LIN {X 0,Y 325.912,Z 530.757,A -85,B 0,C 180,E1 14086.323,E2 14086.323} C_VEL
LIN {X 0,Y 331.424,Z 417.148,A -85,B 0,C 180,E1 14083.968,E2 14083.968} C_VEL
LIN {X 0,Y 322.089,Z 400.841,A -85,B 0,C 180,E1 14081.452,E2 14081.452} C_VEL
LIN {X 0,Y 313.138,Z 386.861,A -85,B 0,C 180,E1 14078.803,E2 14078.803} C_VEL
LIN {X 0,Y 303.548,Z 373.217,A -85,B 0,C 180,E1 14075.606,E2 14075.606} C_VEL
LIN {X 0,Y 293.892,Z 360.856,A -85,B 0,C 180,E1 14071.883,E2 14071.883} C_VEL
LIN {X 0,Y 289.242,Z 355.015,A -85,B 0,C 180,E1 14069.74,E2 14069.74} C_VEL
LIN {X 0,Y 286.141,Z 348.999,A -85,B 0,C 180,E1 14066.345,E2 14066.345} C_VEL
LIN {X 0,Y 283.721,Z 344.309,A -85,B 0,C 180,E1 14063.248,E2 14063.248} C_VEL
LIN {X 0,Y 281.408,Z 340.402,A -85,B 0,C 180,E1 14059.944,E2 14059.944} C_VEL
LIN {X 0,Y 280.7,Z 339.051,A -85,B 0,C 180,E1 14058.699,E2 14058.699} C_VEL
LIN {X 0,Y 277.789,Z 333.962,A -85,B 0,C 180,E1 14052.05,E2 14052.05} C_VEL
LIN {X 0,Y 276.387,Z 332.628,A -85,B 0,C 180,E1 14046.439,E2 14046.439} C_VEL
LIN {X 0,Y 276.572,Z 332.801,A -85,B 0,C 180,E1 14041.243,E2 14041.243} C_VEL
LIN {X 0,Y 278.076,Z 334.319,A -85,B 0,C 180,E1 14036.29,E2 14036.29} C_VEL
LIN {X 0,Y 281.635,Z 340.034,A -85,B 0,C 180,E1 14029.362,E2 14029.362} C_VEL
LIN {X 0,Y 283.845,Z 344.262,A -85,B 0,C 180,E1 14026.141,E2 14026.141} C_VEL
LIN {X 0,Y 284.804,Z 345.431,A -85,B 0,C 180,E1 14025.151,E2 14025.151} C_VEL
LIN {X 0,Y 287.071,Z 349.665,A -85,B 0,C 180,E1 14022.571,E2 14022.571} C_VEL
LIN {X 0,Y 287.875,Z 350.984,A -85,B 0,C 180,E1 14021.785,E2 14021.785} C_VEL
LIN {X 0,Y 290.746,Z 356.23,A -85,B 0,C 180,E1 14019.044,E2 14019.044} C_VEL
LIN {X 0,Y 293.325,Z 361.286,A -85,B 0,C 180,E1 14016.709,E2 14016.709} C_VEL
LIN {X 0,Y 297.429,Z 368.871,A -85,B 0,C 180,E1 14013.658,E2 14013.658} C_VEL
LIN {X 0,Y 299.486,Z 372.66,A -85,B 0,C 180,E1 14012.405,E2 14012.405} C_VEL
LIN {X 0,Y 308.932,Z 386.315,A -85,B 0,C 180,E1 14009.029,E2 14009.029} C_VEL
LIN {X 0,Y 317.812,Z 400.47,A -85,B 0,C 180,E1 14006.216,E2 14006.216} C_VEL
LIN {X 0,Y 327.251,Z 417.04,A -85,B 0,C 180,E1 14003.513,E2 14003.513} C_VEL
LIN {X 0,Y 331.466,Z 425.611,A -85,B 0,C 180,E1 14002.357,E2 14002.357} C_VEL
LIN {X 0,Y 331.933,Z 439.03,A -85,B 0,C 180,E1 14001.807,E2 14001.807} C_VEL
LIN {X 0,Y 321.091,Z 624.81,A -85,B 0,C 180,E1 13997.585,E2 13997.585} C_VEL
LIN {X 0,Y 318.521,Z 646.616,A -85,B 0,C 180,E1 13996.819,E2 13996.819} C_VEL
LIN {X 0,Y 314.877,Z 667.549,A -85,B 0,C 180,E1 13995.793,E2 13995.793} C_VEL
LIN {X 0,Y 310.481,Z 687.705,A -85,B 0,C 180,E1 13994.459,E2 13994.459} C_VEL
LIN {X 0,Y 305.511,Z 707.389,A -85,B 0,C 180,E1 13992.755,E2 13992.755} C_VEL
LIN {X 0,Y 300.341,Z 725.782,A -85,B 0,C 180,E1 13990.729,E2 13990.729} C_VEL
LIN {X 0,Y 295.179,Z 742.727,A -85,B 0,C 180,E1 13988.414,E2 13988.414} C_VEL
LIN {X 0,Y 290.123,Z 758.694,A -85,B 0,C 180,E1 13985.742,E2 13985.742} C_VEL
LIN {X 0,Y 285.541,Z 773.07,A -85,B 0,C 180,E1 13982.819,E2 13982.819} C_VEL
LIN {X 0,Y 281.238,Z 787.006,A -85,B 0,C 180,E1 13979.38,E2 13979.38} C_VEL
LIN {X 0,Y 277.714,Z 799.537,A -85,B 0,C 180,E1 13975.596,E2 13975.596} C_VEL
LIN {X 0,Y 275.265,Z 809.934,A -85,B 0,C 180,E1 13971.746,E2 13971.746} C_VEL
LIN {X 0,Y 273.777,Z 818.455,A -85,B 0,C 180,E1 13967.864,E2 13967.864} C_VEL
LIN {X 0,Y 273.13,Z 825.558,A -85,B 0,C 180,E1 13963.765,E2 13963.765} C_VEL
LIN {X 0,Y 273.196,Z 830.779,A -85,B 0,C 180,E1 13959.692,E2 13959.692} C_VEL
LIN {X 0,Y 273.612,Z 834.096,A -85,B 0,C 180,E1 13955.873,E2 13955.873} C_VEL
LIN {X 0,Y 273.979,Z 835.824,A -85,B 0,C 180,E1 13952.301,E2 13952.301} C_VEL
LIN {X 0,Y 274.057,Z 836.01,A -85,B 0,C 180,E1 13948.955,E2 13948.955} C_VEL
LIN {X 0,Y 273.763,Z 834.896,A -85,B 0,C 180,E1 13945.391,E2 13945.391} C_VEL
LIN {X 0,Y 273.337,Z 832.235,A -85,B 0,C 180,E1 13941.798,E2 13941.798} C_VEL
LIN {X 0,Y 273.084,Z 827.633,A -85,B 0,C 180,E1 13937.74,E2 13937.74} C_VEL
LIN {X 0,Y 273.452,Z 821.244,A -85,B 0,C 180,E1 13933.648,E2 13933.648} C_VEL
LIN {X 0,Y 274.661,Z 812.965,A -85,B 0,C 180,E1 13929.546,E2 13929.546} C_VEL
LIN {X 0,Y 276.918,Z 802.631,A -85,B 0,C 180,E1 13925.467,E2 13925.467} C_VEL
LIN {X 0,Y 280.149,Z 790.716,A -85,B 0,C 180,E1 13921.662,E2 13921.662} C_VEL
LIN {X 0,Y 284.213,Z 777.257,A -85,B 0,C 180,E1 13918.151,E2 13918.151} C_VEL
LIN {X 0,Y 288.798,Z 762.744,A -85,B 0,C 180,E1 13915.043,E2 13915.043} C_VEL
LIN {X 0,Y 293.673,Z 747.357,A -85,B 0,C 180,E1 13912.329,E2 13912.329} C_VEL
LIN {X 0,Y 298.826,Z 730.575,A -85,B 0,C 180,E1 13909.903,E2 13909.903} C_VEL
LIN {X 0,Y 304.127,Z 712.146,A -85,B 0,C 180,E1 13907.755,E2 13907.755} C_VEL
LIN {X 0,Y 309.042,Z 693.226,A -85,B 0,C 180,E1 13906.004,E2 13906.004} C_VEL
LIN {X 0,Y 313.618,Z 673.067,A -85,B 0,C 180,E1 13904.559,E2 13904.559} C_VEL
LIN {X 0,Y 317.514,Z 652.33,A -85,B 0,C 180,E1 13903.454,E2 13903.454} C_VEL
LIN {X 0,Y 320.333,Z 631.352,A -85,B 0,C 180,E1 13902.639,E2 13902.639} C_VEL
LIN {X 0,Y 322.11,Z 608.021,A -85,B 0,C 180,E1 13902.015,E2 13902.015} C_VEL
LIN {X 0,Y 331.889,Z 436.421,A -85,B 0,C 180,E1 13898.133,E2 13898.133} C_VEL
LIN {X 0,Y 331.118,Z 424.68,A -85,B 0,C 180,E1 13897.587,E2 13897.587} C_VEL
LIN {X 0,Y 322.829,Z 409.225,A -85,B 0,C 180,E1 13895.31,E2 13895.31} C_VEL
LIN {X 0,Y 314.205,Z 394.789,A -85,B 0,C 180,E1 13892.749,E2 13892.749} C_VEL
LIN {X 0,Y 306.355,Z 382.678,A -85,B 0,C 180,E1 13890.173,E2 13890.173} C_VEL
LIN {X 0,Y 298.711,Z 371.628,A -85,B 0,C 180,E1 13887.349,E2 13887.349} C_VEL
LIN {X 0,Y 294.503,Z 363.438,A -85,B 0,C 180,E1 13884.255,E2 13884.255} C_VEL
LIN {X 0,Y 291.847,Z 358.564,A -85,B 0,C 180,E1 13882.139,E2 13882.139} C_VEL
LIN {X 0,Y 289.754,Z 354.487,A -85,B 0,C 180,E1 13880.186,E2 13880.186} C_VEL
LIN {X 0,Y 287.159,Z 349.76,A -85,B 0,C 180,E1 13877.633,E2 13877.633} C_VEL
LIN {X 0,Y 284.83,Z 345.563,A -85,B 0,C 180,E1 13875.056,E2 13875.056} C_VEL
LIN {X 0,Y 281.786,Z 340.679,A -85,B 0,C 180,E1 13871.253,E2 13871.253} C_VEL
LIN {X 0,Y 281.192,Z 339.431,A -85,B 0,C 180,E1 13870.241,E2 13870.241} C_VEL
LIN {X 0,Y 277.823,Z 333.98,A -85,B 0,C 180,E1 13863.507,E2 13863.507} C_VEL
LIN {X 0,Y 276.215,Z 332.418,A -85,B 0,C 180,E1 13857.505,E2 13857.505} C_VEL
LIN {X 0,Y 276.38,Z 332.578,A -85,B 0,C 180,E1 13852.098,E2 13852.098} C_VEL
LIN {X 0,Y 277.952,Z 334.225,A -85,B 0,C 180,E1 13846.901,E2 13846.901} C_VEL
LIN {X 0,Y 281.193,Z 339.671,A -85,B 0,C 180,E1 13840.257,E2 13840.257} C_VEL
LIN {X 0,Y 283.306,Z 343.892,A -85,B 0,C 180,E1 13836.936,E2 13836.936} C_VEL
LIN {X 0,Y 284.176,Z 345.216,A -85,B 0,C 180,E1 13835.911,E2 13835.911} C_VEL
LIN {X 0,Y 286.766,Z 350.132,A -85,B 0,C 180,E1 13832.757,E2 13832.757} C_VEL
LIN {X 0,Y 289.262,Z 355.103,A -85,B 0,C 180,E1 13830.034,E2 13830.034} C_VEL
LIN {X 0,Y 295.268,Z 362.715,A -85,B 0,C 180,E1 13827.366,E2 13827.366} C_VEL
LIN {X 0,Y 303.925,Z 373.809,A -85,B 0,C 180,E1 13824.097,E2 13824.097} C_VEL
LIN {X 0,Y 313.853,Z 387.94,A -85,B 0,C 180,E1 13820.833,E2 13820.833} C_VEL
LIN {X 0,Y 323.057,Z 402.598,A -85,B 0,C 180,E1 13818.136,E2 13818.136} C_VEL
LIN {X 0,Y 331.436,Z 417.301,A -85,B 0,C 180,E1 13815.892,E2 13815.892} C_VEL
LIN {X 0,Y 324.029,Z 570.746,A -85,B 0,C 180,E1 13812.693,E2 13812.693} C_VEL
LIN {X 0,Y 322.622,Z 590.161,A -85,B 0,C 180,E1 13812.013,E2 13812.013} C_VEL
LIN {X 0,Y 320.358,Z 608.777,A -85,B 0,C 180,E1 13811.069,E2 13811.069} C_VEL
LIN {X 0,Y 317.4,Z 626.429,A -85,B 0,C 180,E1 13809.869,E2 13809.869} C_VEL
LIN {X 0,Y 313.615,Z 644.125,A -85,B 0,C 180,E1 13808.322,E2 13808.322} C_VEL
LIN {X 0,Y 309.308,Z 660.695,A -85,B 0,C 180,E1 13806.497,E2 13806.497} C_VEL
LIN {X 0,Y 304.53,Z 676.538,A -85,B 0,C 180,E1 13804.313,E2 13804.313} C_VEL
LIN {X 0,Y 299.564,Z 691.068,A -85,B 0,C 180,E1 13801.826,E2 13801.826} C_VEL
LIN {X 0,Y 294.635,Z 704.227,A -85,B 0,C 180,E1 13799.03,E2 13799.03} C_VEL
LIN {X 0,Y 289.962,Z 715.814,A -85,B 0,C 180,E1 13795.971,E2 13795.971} C_VEL
LIN {X 0,Y 285.729,Z 725.888,A -85,B 0,C 180,E1 13792.638,E2 13792.638} C_VEL
LIN {X 0,Y 282.058,Z 734.454,A -85,B 0,C 180,E1 13789.033,E2 13789.033} C_VEL
LIN {X 0,Y 279.071,Z 741.482,A -85,B 0,C 180,E1 13785.161,E2 13785.161} C_VEL
LIN {X 0,Y 276.972,Z 746.671,A -85,B 0,C 180,E1 13781.241,E2 13781.241} C_VEL
LIN {X 0,Y 275.562,Z 750.342,A -85,B 0,C 180,E1 13777.086,E2 13777.086} C_VEL
LIN {X 0,Y 274.872,Z 752.306,A -85,B 0,C 180,E1 13772.919,E2 13772.919} C_VEL
LIN {X 0,Y 274.762,Z 752.649,A -85,B 0,C 180,E1 13768.749,E2 13768.749} C_VEL
LIN {X 0,Y 275.198,Z 751.384,A -85,B 0,C 180,E1 13764.572,E2 13764.572} C_VEL
LIN {X 0,Y 276.288,Z 748.463,A -85,B 0,C 180,E1 13760.418,E2 13760.418} C_VEL
LIN {X 0,Y 278.158,Z 743.76,A -85,B 0,C 180,E1 13756.277,E2 13756.277} C_VEL
LIN {X 0,Y 280.792,Z 737.489,A -85,B 0,C 180,E1 13752.382,E2 13752.382} C_VEL
LIN {X 0,Y 284.139,Z 729.734,A -85,B 0,C 180,E1 13748.75,E2 13748.75} C_VEL
LIN {X 0,Y 288.037,Z 720.554,A -85,B 0,C 180,E1 13745.384,E2 13745.384} C_VEL
LIN {X 0,Y 292.411,Z 709.978,A -85,B 0,C 180,E1 13742.289,E2 13742.289} C_VEL
LIN {X 0,Y 297.09,Z 698.005,A -85,B 0,C 180,E1 13739.458,E2 13739.458} C_VEL
LIN {X 0,Y 302.111,Z 684.038,A -85,B 0,C 180,E1 13736.789,E2 13736.789} C_VEL
LIN {X 0,Y 307.017,Z 668.867,A -85,B 0,C 180,E1 13734.458,E2 13734.458} C_VEL
LIN {X 0,Y 311.62,Z 652.509,A -85,B 0,C 180,E1 13732.438,E2 13732.438} C_VEL
LIN {X 0,Y 315.588,Z 635.868,A -85,B 0,C 180,E1 13730.799,E2 13730.799} C_VEL
LIN {X 0,Y 318.977,Z 618.266,A -85,B 0,C 180,E1 13729.428,E2 13729.428} C_VEL
LIN {X 0,Y 321.711,Z 599.435,A -85,B 0,C 180,E1 13728.312,E2 13728.312} C_VEL
LIN {X 0,Y 323.578,Z 579.916,A -85,B 0,C 180,E1 13727.482,E2 13727.482} C_VEL
LIN {X 0,Y 324.743,Z 555.923,A -85,B 0,C 180,E1 13726.846,E2 13726.846} C_VEL
LIN {X 0,Y 325.912,Z 530.757,A -85,B 0,C 180,E1 13726.323,E2 13726.323} C_VEL
LIN {X 0,Y 325.598,Z 523.167,A -85,B 0,C 180,E1 13726.039,E2 13726.039} C_VEL
LIN {X 0,Y 322.366,Z 503.342,A -85,B 0,C 180,E1 13724.812,E2 13724.812} C_VEL
LIN {X 0,Y 322.193,Z 496.817,A -85,B 0,C 180,E1 13724.576,E2 13724.576} C_VEL
LIN {X 0,Y 326.056,Z 420.531,A -85,B 0,C 180,E1 13722.97,E2 13722.97} C_VEL
LIN {X 0,Y 317.729,Z 405.913,A -85,B 0,C 180,E1 13720.619,E2 13720.619} C_VEL
LIN {X 0,Y 309.549,Z 392.937,A -85,B 0,C 180,E1 13718.093,E2 13718.093} C_VEL
LIN {X 0,Y 300.513,Z 379.839,A -85,B 0,C 180,E1 13714.968,E2 13714.968} C_VEL
LIN {X 0,Y 291.185,Z 367.626,A -85,B 0,C 180,E1 13711.232,E2 13711.232} C_VEL
LIN {X 0,Y 285.424,Z 360.648,A -85,B 0,C 180,E1 13708.566,E2 13708.566} C_VEL
LIN {X 0,Y 281.908,Z 356.155,A -85,B 0,C 180,E1 13706.651,E2 13706.651} C_VEL
LIN {X 0,Y 279.002,Z 350.696,A -85,B 0,C 180,E1 13702.93,E2 13702.93} C_VEL
LIN {X 0,Y 276.761,Z 346.463,A -85,B 0,C 180,E1 13699.413,E2 13699.413} C_VEL
LIN {X 0,Y 273.571,Z 340.764,A -85,B 0,C 180,E1 13692.025,E2 13692.025} C_VEL
LIN {X 0,Y 272.202,Z 339.441,A -85,B 0,C 180,E1 13686.327,E2 13686.327} C_VEL
LIN {X 0,Y 272.456,Z 339.661,A -85,B 0,C 180,E1 13681.262,E2 13681.262} C_VEL
LIN {X 0,Y 273.881,Z 341.096,A -85,B 0,C 180,E1 13676.442,E2 13676.442} C_VEL
LIN {X 0,Y 277.267,Z 346.64,A -85,B 0,C 180,E1 13669.613,E2 13669.613} C_VEL
LIN {X 0,Y 279.445,Z 350.884,A -85,B 0,C 180,E1 13666.341,E2 13666.341} C_VEL
LIN {X 0,Y 280.36,Z 352.123,A -85,B 0,C 180,E1 13665.333,E2 13665.333} C_VEL
LIN {X 0,Y 282.589,Z 356.255,A -85,B 0,C 180,E1 13662.71,E2 13662.71} C_VEL
LIN {X 0,Y 285.907,Z 362.472,A -85,B 0,C 180,E1 13659.317,E2 13659.317} C_VEL
LIN {X 0,Y 288.869,Z 368.159,A -85,B 0,C 180,E1 13656.76,E2 13656.76} C_VEL
LIN {X 0,Y 290.863,Z 371.534,A -85,B 0,C 180,E1 13655.422,E2 13655.422} C_VEL
LIN {X 0,Y 298.308,Z 382.017,A -85,B 0,C 180,E1 13652.341,E2 13652.341} C_VEL
LIN {X 0,Y 306.047,Z 393.465,A -85,B 0,C 180,E1 13649.523,E2 13649.523} C_VEL
LIN {X 0,Y 314.219,Z 406.761,A -85,B 0,C 180,E1 13646.845,E2 13646.845} C_VEL
LIN {X 0,Y 323.159,Z 422.766,A -85,B 0,C 180,E1 13644.186,E2 13644.186} C_VEL
LIN {X 0,Y 326.324,Z 429.459,A -85,B 0,C 180,E1 13643.27,E2 13643.27} C_VEL
LIN {X 0,Y 326.603,Z 440.209,A -85,B 0,C 180,E1 13642.833,E2 13642.833} C_VEL
LIN {X 0,Y 315.481,Z 623.904,A -85,B 0,C 180,E1 13638.626,E2 13638.626} C_VEL
LIN {X 0,Y 312.841,Z 645.686,A -85,B 0,C 180,E1 13637.856,E2 13637.856} C_VEL
LIN {X 0,Y 309.118,Z 666.476,A -85,B 0,C 180,E1 13636.834,E2 13636.834} C_VEL
LIN {X 0,Y 304.704,Z 686.073,A -85,B 0,C 180,E1 13635.536,E2 13635.536} C_VEL
LIN {X 0,Y 299.76,Z 704.977,A -85,B 0,C 180,E1 13633.907,E2 13633.907} C_VEL
LIN {X 0,Y 294.582,Z 722.809,A -85,B 0,C 180,E1 13631.961,E2 13631.961} C_VEL
LIN {X 0,Y 289.168,Z 739.981,A -85,B 0,C 180,E1 13629.637,E2 13629.637} C_VEL
LIN {X 0,Y 283.936,Z 755.721,A -85,B 0,C 180,E1 13627.024,E2 13627.024} C_VEL
LIN {X 0,Y 278.946,Z 770.642,A -85,B 0,C 180,E1 13623.997,E2 13623.997} C_VEL
LIN {X 0,Y 274.482,Z 784.174,A -85,B 0,C 180,E1 13620.661,E2 13620.661} C_VEL
LIN {X 0,Y 270.765,Z 796.349,A -85,B 0,C 180,E1 13617.013,E2 13617.013} C_VEL
LIN {X 0,Y 267.921,Z 807.109,A -85,B 0,C 180,E1 13613.069,E2 13613.069} C_VEL
LIN {X 0,Y 266.005,Z 816.654,A -85,B 0,C 180,E1 13608.7,E2 13608.7} C_VEL
LIN {X 0,Y 265.206,Z 823.96,A -85,B 0,C 180,E1 13604.408,E2 13604.408} C_VEL
LIN {X 0,Y 265.204,Z 829.303,A -85,B 0,C 180,E1 13600.206,E2 13600.206} C_VEL
LIN {X 0,Y 265.626,Z 832.742,A -85,B 0,C 180,E1 13596.267,E2 13596.267} C_VEL
LIN {X 0,Y 266.028,Z 834.465,A -85,B 0,C 180,E1 13592.8,E2 13592.8} C_VEL
LIN {X 0,Y 266.157,Z 834.862,A -85,B 0,C 180,E1 13589.354,E2 13589.354} C_VEL
LIN {X 0,Y 265.922,Z 834.045,A -85,B 0,C 180,E1 13586.119,E2 13586.119} C_VEL
LIN {X 0,Y 265.435,Z 831.58,A -85,B 0,C 180,E1 13582.206,E2 13582.206} C_VEL
LIN {X 0,Y 265.12,Z 827.563,A -85,B 0,C 180,E1 13578.25,E2 13578.25} C_VEL
LIN {X 0,Y 265.396,Z 821.493,A -85,B 0,C 180,E1 13574.037,E2 13574.037} C_VEL
LIN {X 0,Y 266.529,Z 813.563,A -85,B 0,C 180,E1 13569.811,E2 13569.811} C_VEL
LIN {X 0,Y 268.637,Z 804.049,A -85,B 0,C 180,E1 13565.766,E2 13565.766} C_VEL
LIN {X 0,Y 271.757,Z 792.882,A -85,B 0,C 180,E1 13561.905,E2 13561.905} C_VEL
LIN {X 0,Y 275.768,Z 780.085,A -85,B 0,C 180,E1 13558.284,E2 13558.284} C_VEL
LIN {X 0,Y 280.514,Z 765.839,A -85,B 0,C 180,E1 13554.981,E2 13554.981} C_VEL
LIN {X 0,Y 285.698,Z 750.379,A -85,B 0,C 180,E1 13552.046,E2 13552.046} C_VEL
LIN {X 0,Y 291.038,Z 734.033,A -85,B 0,C 180,E1 13549.512,E2 13549.512} C_VEL
LIN {X 0,Y 296.423,Z 716.509,A -85,B 0,C 180,E1 13547.315,E2 13547.315} C_VEL
LIN {X 0,Y 301.818,Z 697.169,A -85,B 0,C 180,E1 13545.389,E2 13545.389} C_VEL
LIN {X 0,Y 306.581,Z 677.71,A -85,B 0,C 180,E1 13543.885,E2 13543.885} C_VEL
LIN {X 0,Y 310.665,Z 657.913,A -85,B 0,C 180,E1 13542.727,E2 13542.727} C_VEL
LIN {X 0,Y 313.859,Z 637.577,A -85,B 0,C 180,E1 13541.847,E2 13541.847} C_VEL
LIN {X 0,Y 315.922,Z 616.704,A -85,B 0,C 180,E1 13541.203,E2 13541.203} C_VEL
LIN {X 0,Y 326.575,Z 437.654,A -85,B 0,C 180,E1 13537.112,E2 13537.112} C_VEL
LIN {X 0,Y 326.002,Z 428.555,A -85,B 0,C 180,E1 13536.677,E2 13536.677} C_VEL
LIN {X 0,Y 317.855,Z 413.201,A -85,B 0,C 180,E1 13534.323,E2 13534.323} C_VEL
LIN {X 0,Y 308.899,Z 398.062,A -85,B 0,C 180,E1 13531.517,E2 13531.517} C_VEL
LIN {X 0,Y 300.403,Z 384.981,A -85,B 0,C 180,E1 13528.53,E2 13528.53} C_VEL
LIN {X 0,Y 292.847,Z 374.376,A -85,B 0,C 180,E1 13525.534,E2 13525.534} C_VEL
LIN {X 0,Y 290.063,Z 370.213,A -85,B 0,C 180,E1 13524.217,E2 13524.217} C_VEL
LIN {X 0,Y 286.914,Z 364.504,A -85,B 0,C 180,E1 13521.678,E2 13521.678} C_VEL
LIN {X 0,Y 284.984,Z 360.764,A -85,B 0,C 180,E1 13519.896,E2 13519.896} C_VEL
LIN {X 0,Y 282.411,Z 356.076,A -85,B 0,C 180,E1 13517.301,E2 13517.301} C_VEL
LIN {X 0,Y 279.905,Z 351.338,A -85,B 0,C 180,E1 13514.269,E2 13514.269} C_VEL
LIN {X 0,Y 277.516,Z 347.594,A -85,B 0,C 180,E1 13511.218,E2 13511.218} C_VEL
LIN {X 0,Y 276.813,Z 346.091,A -85,B 0,C 180,E1 13509.984,E2 13509.984} C_VEL
LIN {X 0,Y 273.63,Z 340.766,A -85,B 0,C 180,E1 13503.351,E2 13503.351} C_VEL
LIN {X 0,Y 272.02,Z 339.216,A -85,B 0,C 180,E1 13497.261,E2 13497.261} C_VEL
LIN {X 0,Y 272.217,Z 339.429,A -85,B 0,C 180,E1 13491.976,E2 13491.976} C_VEL
LIN {X 0,Y 273.675,Z 341.008,A -85,B 0,C 180,E1 13486.908,E2 13486.908} C_VEL
LIN {X 0,Y 276.735,Z 346.396,A -85,B 0,C 180,E1 13480.365,E2 13480.365} C_VEL
LIN {X 0,Y 278.871,Z 350.546,A -85,B 0,C 180,E1 13476.995,E2 13476.995} C_VEL
LIN {X 0,Y 279.602,Z 351.984,A -85,B 0,C 180,E1 13475.941,E2 13475.941} C_VEL
LIN {X 0,Y 282.03,Z 356.488,A -85,B 0,C 180,E1 13473.012,E2 13473.012} C_VEL
LIN {X 0,Y 285.873,Z 361.055,A -85,B 0,C 180,E1 13471.026,E2 13471.026} C_VEL
LIN {X 0,Y 292.839,Z 369.89,A -85,B 0,C 180,E1 13467.873,E2 13467.873} C_VEL
LIN {X 0,Y 300.999,Z 380.593,A -85,B 0,C 180,E1 13464.69,E2 13464.69} C_VEL
LIN {X 0,Y 310.626,Z 394.567,A -85,B 0,C 180,E1 13461.416,E2 13461.416} C_VEL
LIN {X 0,Y 319.403,Z 408.86,A -85,B 0,C 180,E1 13458.75,E2 13458.75} C_VEL
LIN {X 0,Y 326.078,Z 420.895,A -85,B 0,C 180,E1 13456.879,E2 13456.879} C_VEL
LIN {X 0,Y 318.463,Z 571.358,A -85,B 0,C 180,E1 13453.711,E2 13453.711} C_VEL
LIN {X 0,Y 316.99,Z 590.894,A -85,B 0,C 180,E1 13453.022,E2 13453.022} C_VEL
LIN {X 0,Y 314.593,Z 609.838,A -85,B 0,C 180,E1 13452.052,E2 13452.052} C_VEL
LIN {X 0,Y 311.344,Z 628.339,A -85,B 0,C 180,E1 13450.771,E2 13450.771} C_VEL
LIN {X 0,Y 307.479,Z 645.583,A -85,B 0,C 180,E1 13449.232,E2 13449.232} C_VEL
LIN {X 0,Y 303.009,Z 662.069,A -85,B 0,C 180,E1 13447.383,E2 13447.383} C_VEL
LIN {X 0,Y 298.164,Z 677.501,A -85,B 0,C 180,E1 13445.223,E2 13445.223} C_VEL
LIN {X 0,Y 293.241,Z 691.381,A -85,B 0,C 180,E1 13442.828,E2 13442.828} C_VEL
LIN {X 0,Y 288.068,Z 704.681,A -85,B 0,C 180,E1 13439.987,E2 13439.987} C_VEL
LIN {X 0,Y 283.147,Z 716.394,A -85,B 0,C 180,E1 13436.871,E2 13436.871} C_VEL
LIN {X 0,Y 278.666,Z 726.58,A -85,B 0,C 180,E1 13433.469,E2 13433.469} C_VEL
LIN {X 0,Y 274.765,Z 735.247,A -85,B 0,C 180,E1 13429.78,E2 13429.78} C_VEL
LIN {X 0,Y 271.565,Z 742.37,A -85,B 0,C 180,E1 13425.81,E2 13425.81} C_VEL
LIN {X 0,Y 269.2,Z 747.878,A -85,B 0,C 180,E1 13421.57,E2 13421.57} C_VEL
LIN {X 0,Y 267.705,Z 751.546,A -85,B 0,C 180,E1 13417.295,E2 13417.295} C_VEL
LIN {X 0,Y 266.971,Z 753.508,A -85,B 0,C 180,E1 13413.006,E2 13413.006} C_VEL
LIN {X 0,Y 266.854,Z 753.851,A -85,B 0,C 180,E1 13408.712,E2 13408.712} C_VEL
LIN {X 0,Y 267.317,Z 752.59,A -85,B 0,C 180,E1 13404.419,E2 13404.419} C_VEL
LIN {X 0,Y 268.477,Z 749.667,A -85,B 0,C 180,E1 13400.136,E2 13400.136} C_VEL
LIN {X 0,Y 270.459,Z 744.967,A -85,B 0,C 180,E1 13395.878,E2 13395.878} C_VEL
LIN {X 0,Y 273.239,Z 738.7,A -85,B 0,C 180,E1 13391.879,E2 13391.879} C_VEL
LIN {X 0,Y 276.759,Z 730.951,A -85,B 0,C 180,E1 13388.155,E2 13388.155} C_VEL
LIN {X 0,Y 280.849,Z 721.782,A -85,B 0,C 180,E1 13384.71,E2 13384.71} C_VEL
LIN {X 0,Y 285.424,Z 711.219,A -85,B 0,C 180,E1 13381.549,E2 13381.549} C_VEL
LIN {X 0,Y 290.65,Z 698.387,A -85,B 0,C 180,E1 13378.475,E2 13378.475} C_VEL
LIN {X 0,Y 295.722,Z 684.799,A -85,B 0,C 180,E1 13375.858,E2 13375.858} C_VEL
LIN {X 0,Y 300.837,Z 669.56,A -85,B 0,C 180,E1 13373.494,E2 13373.494} C_VEL
LIN {X 0,Y 305.413,Z 653.91,A -85,B 0,C 180,E1 13371.538,E2 13371.538} C_VEL
LIN {X 0,Y 309.751,Z 636.388,A -85,B 0,C 180,E1 13369.792,E2 13369.792} C_VEL
LIN {X 0,Y 313.272,Z 618.661,A -85,B 0,C 180,E1 13368.406,E2 13368.406} C_VEL
LIN {X 0,Y 316.124,Z 599.539,A -85,B 0,C 180,E1 13367.272,E2 13367.272} C_VEL
LIN {X 0,Y 318.041,Z 579.955,A -85,B 0,C 180,E1 13366.444,E2 13366.444} C_VEL
LIN {X 0,Y 319.275,Z 555.252,A -85,B 0,C 180,E1 13365.793,E2 13365.793} C_VEL
LIN {X 0,Y 322.193,Z 496.817,A -85,B 0,C 180,E1 13364.576,E2 13364.576} C_VEL
LIN {X 0,Y 321.919,Z 489.23,A -85,B 0,C 180,E1 13364.285,E2 13364.285} C_VEL
LIN {X 0,Y 318.902,Z 469.415,A -85,B 0,C 180,E1 13363.023,E2 13363.023} C_VEL
LIN {X 0,Y 318.781,Z 462.892,A -85,B 0,C 180,E1 13362.784,E2 13362.784} C_VEL
LIN {X 0,Y 320.861,Z 424.086,A -85,B 0,C 180,E1 13361.958,E2 13361.958} C_VEL
LIN {X 0,Y 312.608,Z 409.503,A -85,B 0,C 180,E1 13359.501,E2 13359.501} C_VEL
LIN {X 0,Y 303.827,Z 395.623,A -85,B 0,C 180,E1 13356.618,E2 13356.618} C_VEL
LIN {X 0,Y 295.497,Z 383.738,A -85,B 0,C 180,E1 13353.531,E2 13353.531} C_VEL
LIN {X 0,Y 287.709,Z 373.406,A -85,B 0,C 180,E1 13350.202,E2 13350.202} C_VEL
LIN {X 0,Y 282.994,Z 367.663,A -85,B 0,C 180,E1 13347.914,E2 13347.914} C_VEL
LIN {X 0,Y 278.943,Z 362.711,A -85,B 0,C 180,E1 13345.704,E2 13345.704} C_VEL
LIN {X 0,Y 275.103,Z 358.176,A -85,B 0,C 180,E1 13343.339,E2 13343.339} C_VEL
LIN {X 0,Y 274.001,Z 356.757,A -85,B 0,C 180,E1 13342.304,E2 13342.304} C_VEL
LIN {X 0,Y 272.017,Z 352.491,A -85,B 0,C 180,E1 13338.651,E2 13338.651} C_VEL
LIN {X 0,Y 269.226,Z 347.427,A -85,B 0,C 180,E1 13331.787,E2 13331.787} C_VEL
LIN {X 0,Y 268.004,Z 346.218,A -85,B 0,C 180,E1 13325.782,E2 13325.782} C_VEL
LIN {X 0,Y 268.413,Z 346.646,A -85,B 0,C 180,E1 13320.641,E2 13320.641} C_VEL
LIN {X 0,Y 269.761,Z 347.998,A -85,B 0,C 180,E1 13316.388,E2 13316.388} C_VEL
LIN {X 0,Y 272.967,Z 353.552,A -85,B 0,C 180,E1 13309.661,E2 13309.661} C_VEL
LIN {X 0,Y 275.149,Z 357.655,A -85,B 0,C 180,E1 13306.338,E2 13306.338} C_VEL
LIN {X 0,Y 275.934,Z 359.08,A -85,B 0,C 180,E1 13305.307,E2 13305.307} C_VEL
LIN {X 0,Y 278.607,Z 363.943,A -85,B 0,C 180,E1 13302.239,E2 13302.239} C_VEL
LIN {X 0,Y 281.536,Z 369.341,A -85,B 0,C 180,E1 13299.416,E2 13299.416} C_VEL
LIN {X 0,Y 288.409,Z 378.688,A -85,B 0,C 180,E1 13295.962,E2 13295.962} C_VEL
LIN {X 0,Y 295.489,Z 388.867,A -85,B 0,C 180,E1 13292.928,E2 13292.928} C_VEL
LIN {X 0,Y 302.956,Z 400.202,A -85,B 0,C 180,E1 13290.109,E2 13290.109} C_VEL
LIN {X 0,Y 310.665,Z 413.045,A -85,B 0,C 180,E1 13287.488,E2 13287.488} C_VEL
LIN {X 0,Y 319.096,Z 428.488,A -85,B 0,C 180,E1 13284.875,E2 13284.875} C_VEL
LIN {X 0,Y 321.258,Z 433.222,A -85,B 0,C 180,E1 13284.217,E2 13284.217} C_VEL
LIN {X 0,Y 321.382,Z 441.415,A -85,B 0,C 180,E1 13283.892,E2 13283.892} C_VEL
LIN {X 0,Y 309.98,Z 622.999,A -85,B 0,C 180,E1 13279.705,E2 13279.705} C_VEL
LIN {X 0,Y 307.28,Z 644.682,A -85,B 0,C 180,E1 13278.935,E2 13278.935} C_VEL
LIN {X 0,Y 303.47,Z 665.368,A -85,B 0,C 180,E1 13277.916,E2 13277.916} C_VEL
LIN {X 0,Y 298.765,Z 685.59,A -85,B 0,C 180,E1 13276.569,E2 13276.569} C_VEL
LIN {X 0,Y 293.432,Z 705.157,A -85,B 0,C 180,E1 13274.856,E2 13274.856} C_VEL
LIN {X 0,Y 287.796,Z 723.659,A -85,B 0,C 180,E1 13272.78,E2 13272.78} C_VEL
LIN {X 0,Y 282.026,Z 741.029,A -85,B 0,C 180,E1 13270.339,E2 13270.339} C_VEL
LIN {X 0,Y 276.407,Z 757.054,A -85,B 0,C 180,E1 13267.554,E2 13267.554} C_VEL
LIN {X 0,Y 271.431,Z 771.124,A -85,B 0,C 180,E1 13264.56,E2 13264.56} C_VEL
LIN {X 0,Y 266.554,Z 785.146,A -85,B 0,C 180,E1 13260.923,E2 13260.923} C_VEL
LIN {X 0,Y 262.573,Z 797.58,A -85,B 0,C 180,E1 13256.945,E2 13256.945} C_VEL
LIN {X 0,Y 259.636,Z 808.401,A -85,B 0,C 180,E1 13252.649,E2 13252.649} C_VEL
LIN {X 0,Y 257.828,Z 817.539,A -85,B 0,C 180,E1 13248.073,E2 13248.073} C_VEL
LIN {X 0,Y 257.177,Z 824.425,A -85,B 0,C 180,E1 13243.603,E2 13243.603} C_VEL
LIN {X 0,Y 257.326,Z 829.321,A -85,B 0,C 180,E1 13239.275,E2 13239.275} C_VEL
LIN {X 0,Y 257.81,Z 832.213,A -85,B 0,C 180,E1 13235.341,E2 13235.341} C_VEL
LIN {X 0,Y 258.192,Z 833.52,A -85,B 0,C 180,E1 13231.775,E2 13231.775} C_VEL
LIN {X 0,Y 258.221,Z 833.577,A -85,B 0,C 180,E1 13228.669,E2 13228.669} C_VEL
LIN {X 0,Y 257.873,Z 832.472,A -85,B 0,C 180,E1 13225.107,E2 13225.107} C_VEL
LIN {X 0,Y 257.392,Z 829.782,A -85,B 0,C 180,E1 13221.286,E2 13221.286} C_VEL
LIN {X 0,Y 257.157,Z 825.142,A -85,B 0,C 180,E1 13216.967,E2 13216.967} C_VEL
LIN {X 0,Y 257.649,Z 818.824,A -85,B 0,C 180,E1 13212.678,E2 13212.678} C_VEL
LIN {X 0,Y 259.172,Z 810.403,A -85,B 0,C 180,E1 13208.263,E2 13208.263} C_VEL
LIN {X 0,Y 261.847,Z 800.038,A -85,B 0,C 180,E1 13203.953,E2 13203.953} C_VEL
LIN {X 0,Y 265.565,Z 788.098,A -85,B 0,C 180,E1 13199.951,E2 13199.951} C_VEL
LIN {X 0,Y 270.179,Z 774.612,A -85,B 0,C 180,E1 13196.283,E2 13196.283} C_VEL
LIN {X 0,Y 275.675,Z 759.061,A -85,B 0,C 180,E1 13192.852,E2 13192.852} C_VEL
LIN {X 0,Y 281.544,Z 742.29,A -85,B 0,C 180,E1 13189.876,E2 13189.876} C_VEL
LIN {X 0,Y 287.32,Z 724.95,A -85,B 0,C 180,E1 13187.403,E2 13187.403} C_VEL
LIN {X 0,Y 292.908,Z 706.657,A -85,B 0,C 180,E1 13185.318,E2 13185.318} C_VEL
LIN {X 0,Y 298.194,Z 687.393,A -85,B 0,C 180,E1 13183.595,E2 13183.595} C_VEL
LIN {X 0,Y 302.716,Z 668.307,A -85,B 0,C 180,E1 13182.282,E2 13182.282} C_VEL
LIN {X 0,Y 306.579,Z 648.218,A -85,B 0,C 180,E1 13181.243,E2 13181.243} C_VEL
LIN {X 0,Y 309.402,Z 627.413,A -85,B 0,C 180,E1 13180.455,E2 13180.455} C_VEL
LIN {X 0,Y 311.513,Z 598.823,A -85,B 0,C 180,E1 13179.718,E2 13179.718} C_VEL
LIN {X 0,Y 321.355,Z 438.503,A -85,B 0,C 180,E1 13176.039,E2 13176.039} C_VEL
LIN {X 0,Y 320.98,Z 432.39,A -85,B 0,C 180,E1 13175.737,E2 13175.737} C_VEL
LIN {X 0,Y 312.401,Z 416.174,A -85,B 0,C 180,E1 13173.127,E2 13173.127} C_VEL
LIN {X 0,Y 303.613,Z 401.378,A -85,B 0,C 180,E1 13170.201,E2 13170.201} C_VEL
LIN {X 0,Y 295.853,Z 389.496,A -85,B 0,C 180,E1 13167.308,E2 13167.308} C_VEL
LIN {X 0,Y 289.927,Z 380.953,A -85,B 0,C 180,E1 13164.826,E2 13164.826} C_VEL
LIN {X 0,Y 286.251,Z 375.895,A -85,B 0,C 180,E1 13163.138,E2 13163.138} C_VEL
LIN {X 0,Y 281.219,Z 368.69,A -85,B 0,C 180,E1 13160.391,E2 13160.391} C_VEL
LIN {X 0,Y 277.967,Z 362.69,A -85,B 0,C 180,E1 13157.155,E2 13157.155} C_VEL
LIN {X 0,Y 275.164,Z 357.679,A -85,B 0,C 180,E1 13153.876,E2 13153.876} C_VEL
LIN {X 0,Y 272.927,Z 353.563,A -85,B 0,C 180,E1 13150.554,E2 13150.554} C_VEL
LIN {X 0,Y 269.521,Z 347.651,A -85,B 0,C 180,E1 13143.402,E2 13143.402} C_VEL
LIN {X 0,Y 267.908,Z 346.09,A -85,B 0,C 180,E1 13137.433,E2 13137.433} C_VEL
LIN {X 0,Y 268.03,Z 346.237,A -85,B 0,C 180,E1 13132.066,E2 13132.066} C_VEL
LIN {X 0,Y 269.456,Z 347.833,A -85,B 0,C 180,E1 13126.917,E2 13126.917} C_VEL
LIN {X 0,Y 272.292,Z 353.128,A -85,B 0,C 180,E1 13120.478,E2 13120.478} C_VEL
LIN {X 0,Y 274.458,Z 357.249,A -85,B 0,C 180,E1 13116.944,E2 13116.944} C_VEL
LIN {X 0,Y 278.958,Z 362.732,A -85,B 0,C 180,E1 13114.069,E2 13114.069} C_VEL
LIN {X 0,Y 285.034,Z 370.137,A -85,B 0,C 180,E1 13110.869,E2 13110.869} C_VEL
LIN {X 0,Y 291.75,Z 378.69,A -85,B 0,C 180,E1 13107.83,E2 13107.83} C_VEL
LIN {X 0,Y 299.601,Z 389.586,A -85,B 0,C 180,E1 13104.735,E2 13104.735} C_VEL
LIN {X 0,Y 307.927,Z 401.985,A -85,B 0,C 180,E1 13101.847,E2 13101.847} C_VEL
LIN {X 0,Y 317.049,Z 417.21,A -85,B 0,C 180,E1 13099.007,E2 13099.007} C_VEL
LIN {X 0,Y 320.808,Z 424.476,A -85,B 0,C 180,E1 13097.903,E2 13097.903} C_VEL
LIN {X 0,Y 313.005,Z 571.897,A -85,B 0,C 180,E1 13094.768,E2 13094.768} C_VEL
LIN {X 0,Y 311.458,Z 591.638,A -85,B 0,C 180,E1 13094.067,E2 13094.067} C_VEL
LIN {X 0,Y 309.037,Z 610.166,A -85,B 0,C 180,E1 13093.114,E2 13093.114} C_VEL
LIN {X 0,Y 305.73,Z 628.487,A -85,B 0,C 180,E1 13091.847,E2 13091.847} C_VEL
LIN {X 0,Y 301.649,Z 646.164,A -85,B 0,C 180,E1 13090.266,E2 13090.266} C_VEL
LIN {X 0,Y 297.002,Z 662.734,A -85,B 0,C 180,E1 13088.397,E2 13088.397} C_VEL
LIN {X 0,Y 291.753,Z 678.821,A -85,B 0,C 180,E1 13086.117,E2 13086.117} C_VEL
LIN {X 0,Y 286.633,Z 692.662,A -85,B 0,C 180,E1 13083.685,E2 13083.685} C_VEL
LIN {X 0,Y 281.243,Z 705.935,A -85,B 0,C 180,E1 13080.792,E2 13080.792} C_VEL
LIN {X 0,Y 276.104,Z 717.629,A -85,B 0,C 180,E1 13077.614,E2 13077.614} C_VEL
LIN {X 0,Y 271.411,Z 727.804,A -85,B 0,C 180,E1 13074.136,E2 13074.136} C_VEL
LIN {X 0,Y 267.314,Z 736.464,A -85,B 0,C 180,E1 13070.356,E2 13070.356} C_VEL
LIN {X 0,Y 263.941,Z 743.582,A -85,B 0,C 180,E1 13066.279,E2 13066.279} C_VEL
LIN {X 0,Y 261.438,Z 749.087,A -85,B 0,C 180,E1 13061.918,E2 13061.918} C_VEL
LIN {X 0,Y 259.852,Z 752.75,A -85,B 0,C 180,E1 13057.517,E2 13057.517} C_VEL
LIN {X 0,Y 259.071,Z 754.711,A -85,B 0,C 180,E1 13053.097,E2 13053.097} C_VEL
LIN {X 0,Y 258.946,Z 755.052,A -85,B 0,C 180,E1 13048.673,E2 13048.673} C_VEL
LIN {X 0,Y 259.439,Z 753.792,A -85,B 0,C 180,E1 13044.249,E2 13044.249} C_VEL
LIN {X 0,Y 260.673,Z 750.871,A -85,B 0,C 180,E1 13039.838,E2 13039.838} C_VEL
LIN {X 0,Y 262.772,Z 746.174,A -85,B 0,C 180,E1 13035.456,E2 13035.456} C_VEL
LIN {X 0,Y 265.709,Z 739.912,A -85,B 0,C 180,E1 13031.347,E2 13031.347} C_VEL
LIN {X 0,Y 269.412,Z 732.169,A -85,B 0,C 180,E1 13027.527,E2 13027.527} C_VEL
LIN {X 0,Y 273.762,Z 722.884,A -85,B 0,C 180,E1 13023.958,E2 13023.958} C_VEL
LIN {X 0,Y 278.809,Z 711.732,A -85,B 0,C 180,E1 13020.575,E2 13020.575} C_VEL
LIN {X 0,Y 283.938,Z 699.648,A -85,B 0,C 180,E1 13017.64,E2 13017.64} C_VEL
LIN {X 0,Y 289.415,Z 685.558,A -85,B 0,C 180,E1 13014.886,E2 13014.886} C_VEL
LIN {X 0,Y 294.534,Z 670.895,A -85,B 0,C 180,E1 13012.581,E2 13012.581} C_VEL
LIN {X 0,Y 299.506,Z 654.524,A -85,B 0,C 180,E1 13010.51,E2 13010.51} C_VEL
LIN {X 0,Y 303.786,Z 637.887,A -85,B 0,C 180,E1 13008.834,E2 13008.834} C_VEL
LIN {X 0,Y 307.442,Z 620.315,A -85,B 0,C 180,E1 13007.434,E2 13007.434} C_VEL
LIN {X 0,Y 310.382,Z 601.677,A -85,B 0,C 180,E1 13006.301,E2 13006.301} C_VEL
LIN {X 0,Y 312.419,Z 582.429,A -85,B 0,C 180,E1 13005.456,E2 13005.456} C_VEL
LIN {X 0,Y 313.657,Z 560.196,A -85,B 0,C 180,E1 13004.83,E2 13004.83} C_VEL
LIN {X 0,Y 318.781,Z 462.892,A -85,B 0,C 180,E1 13002.784,E2 13002.784} C_VEL
LIN {X 0,Y 318.575,Z 455.305,A -85,B 0,C 180,E1 13002.489,E2 13002.489} C_VEL
LIN {X 0,Y 315.809,Z 435.494,A -85,B 0,C 180,E1 13001.194,E2 13001.194} C_VEL
LIN {X 0,Y 315.722,Z 428.972,A -85,B 0,C 180,E1 13000.948,E2 13000.948} C_VEL
LIN {X 0,Y 315.662,Z 427.477,A -85,B 0,C 180,E1 13000.881,E2 13000.881} C_VEL
LIN {X 0,Y 307.347,Z 412.836,A -85,B 0,C 180,E1 12998.268,E2 12998.268} C_VEL
LIN {X 0,Y 300.149,Z 401.392,A -85,B 0,C 180,E1 12995.777,E2 12995.777} C_VEL
LIN {X 0,Y 292.072,Z 389.55,A -85,B 0,C 180,E1 12992.636,E2 12992.636} C_VEL
LIN {X 0,Y 284.605,Z 379.682,A -85,B 0,C 180,E1 12989.289,E2 12989.289} C_VEL
LIN {X 0,Y 280.969,Z 375.046,A -85,B 0,C 180,E1 12987.442,E2 12987.442} C_VEL
LIN {X 0,Y 277.006,Z 370.123,A -85,B 0,C 180,E1 12985.21,E2 12985.21} C_VEL
LIN {X 0,Y 273.074,Z 365.247,A -85,B 0,C 180,E1 12982.68,E2 12982.68} C_VEL
LIN {X 0,Y 268.53,Z 360.386,A -85,B 0,C 180,E1 12979.241,E2 12979.241} C_VEL
LIN {X 0,Y 267.517,Z 359.038,A -85,B 0,C 180,E1 12978.298,E2 12978.298} C_VEL
LIN {X 0,Y 265.017,Z 354.234,A -85,B 0,C 180,E1 12971.756,E2 12971.756} C_VEL
LIN {X 0,Y 263.83,Z 353.036,A -85,B 0,C 180,E1 12965.655,E2 12965.655} C_VEL
LIN {X 0,Y 264.326,Z 353.564,A -85,B 0,C 180,E1 12960.217,E2 12960.217} C_VEL
LIN {X 0,Y 265.573,Z 354.883,A -85,B 0,C 180,E1 12956.331,E2 12956.331} C_VEL
LIN {X 0,Y 268.502,Z 360.09,A -85,B 0,C 180,E1 12949.921,E2 12949.921} C_VEL
LIN {X 0,Y 270.94,Z 364.479,A -85,B 0,C 180,E1 12946.339,E2 12946.339} C_VEL
LIN {X 0,Y 273.615,Z 369.146,A -85,B 0,C 180,E1 12943.44,E2 12943.44} C_VEL
LIN {X 0,Y 279.467,Z 376.816,A -85,B 0,C 180,E1 12939.858,E2 12939.858} C_VEL
LIN {X 0,Y 286.173,Z 386.133,A -85,B 0,C 180,E1 12936.419,E2 12936.419} C_VEL
LIN {X 0,Y 292.702,Z 395.716,A -85,B 0,C 180,E1 12933.527,E2 12933.527} C_VEL
LIN {X 0,Y 300.012,Z 407.122,A -85,B 0,C 180,E1 12930.666,E2 12930.666} C_VEL
LIN {X 0,Y 307.696,Z 420.322,A -85,B 0,C 180,E1 12927.963,E2 12927.963} C_VEL
LIN {X 0,Y 315.333,Z 434.737,A -85,B 0,C 180,E1 12925.502,E2 12925.502} C_VEL
LIN {X 0,Y 316.291,Z 437.142,A -85,B 0,C 180,E1 12925.188,E2 12925.188} C_VEL
LIN {X 0,Y 316.222,Z 443.384,A -85,B 0,C 180,E1 12924.968,E2 12924.968} C_VEL
LIN {X 0,Y 304.593,Z 622.097,A -85,B 0,C 180,E1 12920.822,E2 12920.822} C_VEL
LIN {X 0,Y 301.813,Z 643.788,A -85,B 0,C 180,E1 12920.049,E2 12920.049} C_VEL
LIN {X 0,Y 297.77,Z 665.007,A -85,B 0,C 180,E1 12918.995,E2 12918.995} C_VEL
LIN {X 0,Y 293.03,Z 684.694,A -85,B 0,C 180,E1 12917.673,E2 12917.673} C_VEL
LIN {X 0,Y 287.673,Z 703.642,A -85,B 0,C 180,E1 12916.009,E2 12916.009} C_VEL
LIN {X 0,Y 282.04,Z 721.457,A -85,B 0,C 180,E1 12914.013,E2 12914.013} C_VEL
LIN {X 0,Y 276.168,Z 738.482,A -85,B 0,C 180,E1 12911.631,E2 12911.631} C_VEL
LIN {X 0,Y 270.255,Z 754.629,A -85,B 0,C 180,E1 12908.835,E2 12908.835} C_VEL
LIN {X 0,Y 264.61,Z 769.797,A -85,B 0,C 180,E1 12905.583,E2 12905.583} C_VEL
LIN {X 0,Y 259.425,Z 783.837,A -85,B 0,C 180,E1 12901.87,E2 12901.87} C_VEL
LIN {X 0,Y 255.163,Z 796.286,A -85,B 0,C 180,E1 12897.794,E2 12897.794} C_VEL
LIN {X 0,Y 251.974,Z 807.122,A -85,B 0,C 180,E1 12893.378,E2 12893.378} C_VEL
LIN {X 0,Y 250.049,Z 815.871,A -85,B 0,C 180,E1 12888.898,E2 12888.898} C_VEL
LIN {X 0,Y 249.253,Z 822.73,A -85,B 0,C 180,E1 12884.401,E2 12884.401} C_VEL
LIN {X 0,Y 249.312,Z 827.793,A -85,B 0,C 180,E1 12879.93,E2 12879.93} C_VEL
LIN {X 0,Y 249.832,Z 830.863,A -85,B 0,C 180,E1 12875.742,E2 12875.742} C_VEL
LIN {X 0,Y 250.258,Z 832.286,A -85,B 0,C 180,E1 12872.061,E2 12872.061} C_VEL
LIN {X 0,Y 250.319,Z 832.404,A -85,B 0,C 180,E1 12868.856,E2 12868.856} C_VEL
LIN {X 0,Y 249.956,Z 831.366,A -85,B 0,C 180,E1 12865.181,E2 12865.181} C_VEL
LIN {X 0,Y 249.439,Z 828.746,A -85,B 0,C 180,E1 12861.239,E2 12861.239} C_VEL
LIN {X 0,Y 249.193,Z 824.191,A -85,B 0,C 180,E1 12856.779,E2 12856.779} C_VEL
LIN {X 0,Y 249.74,Z 817.851,A -85,B 0,C 180,E1 12852.286,E2 12852.286} C_VEL
LIN {X 0,Y 251.355,Z 809.631,A -85,B 0,C 180,E1 12847.797,E2 12847.797} C_VEL
LIN {X 0,Y 254.195,Z 799.352,A -85,B 0,C 180,E1 12843.359,E2 12843.359} C_VEL
LIN {X 0,Y 258.116,Z 787.497,A -85,B 0,C 180,E1 12839.249,E2 12839.249} C_VEL
LIN {X 0,Y 262.962,Z 774.122,A -85,B 0,C 180,E1 12835.492,E2 12835.492} C_VEL
LIN {X 0,Y 268.385,Z 759.548,A -85,B 0,C 180,E1 12832.166,E2 12832.166} C_VEL
LIN {X 0,Y 274.179,Z 743.815,A -85,B 0,C 180,E1 12829.251,E2 12829.251} C_VEL
LIN {X 0,Y 280.09,Z 727.014,A -85,B 0,C 180,E1 12826.735,E2 12826.735} C_VEL
LIN {X 0,Y 285.816,Z 709.369,A -85,B 0,C 180,E1 12824.612,E2 12824.612} C_VEL
LIN {X 0,Y 291.483,Z 689.924,A -85,B 0,C 180,E1 12822.773,E2 12822.773} C_VEL
LIN {X 0,Y 296.536,Z 669.888,A -85,B 0,C 180,E1 12821.326,E2 12821.326} C_VEL
LIN {X 0,Y 300.808,Z 648.932,A -85,B 0,C 180,E1 12820.204,E2 12820.204} C_VEL
LIN {X 0,Y 303.908,Z 627.285,A -85,B 0,C 180,E1 12819.364,E2 12819.364} C_VEL
LIN {X 0,Y 306.061,Z 599.729,A -85,B 0,C 180,E1 12818.64,E2 12818.64} C_VEL
LIN {X 0,Y 316.255,Z 439.472,A -85,B 0,C 180,E1 12814.937,E2 12814.937} C_VEL
LIN {X 0,Y 315.971,Z 436.213,A -85,B 0,C 180,E1 12814.749,E2 12814.749} C_VEL
LIN {X 0,Y 308.414,Z 421.704,A -85,B 0,C 180,E1 12812.338,E2 12812.338} C_VEL
LIN {X 0,Y 300.211,Z 407.543,A -85,B 0,C 180,E1 12809.477,E2 12809.477} C_VEL
LIN {X 0,Y 292.84,Z 396.03,A -85,B 0,C 180,E1 12806.624,E2 12806.624} C_VEL
LIN {X 0,Y 287.054,Z 387.519,A -85,B 0,C 180,E1 12804.104,E2 12804.104} C_VEL
LIN {X 0,Y 283.294,Z 382.254,A -85,B 0,C 180,E1 12802.297,E2 12802.297} C_VEL
LIN {X 0,Y 277.653,Z 374.456,A -85,B 0,C 180,E1 12799.238,E2 12799.238} C_VEL
LIN {X 0,Y 273.404,Z 368.944,A -85,B 0,C 180,E1 12796.573,E2 12796.573} C_VEL
LIN {X 0,Y 270.804,Z 364.328,A -85,B 0,C 180,E1 12793.668,E2 12793.668} C_VEL
LIN {X 0,Y 268.482,Z 360.116,A -85,B 0,C 180,E1 12790.297,E2 12790.297} C_VEL
LIN {X 0,Y 265.269,Z 354.401,A -85,B 0,C 180,E1 12783.241,E2 12783.241} C_VEL
LIN {X 0,Y 263.711,Z 352.868,A -85,B 0,C 180,E1 12776.957,E2 12776.957} C_VEL
LIN {X 0,Y 263.979,Z 353.221,A -85,B 0,C 180,E1 12771.285,E2 12771.285} C_VEL
LIN {X 0,Y 265.225,Z 354.68,A -85,B 0,C 180,E1 12766.927,E2 12766.927} C_VEL
LIN {X 0,Y 267.657,Z 359.152,A -85,B 0,C 180,E1 12761.26,E2 12761.26} C_VEL
LIN {X 0,Y 272.055,Z 364.369,A -85,B 0,C 180,E1 12757.756,E2 12757.756} C_VEL
LIN {X 0,Y 273.384,Z 365.807,A -85,B 0,C 180,E1 12756.848,E2 12756.848} C_VEL
LIN {X 0,Y 277.358,Z 370.442,A -85,B 0,C 180,E1 12754.367,E2 12754.367} C_VEL
LIN {X 0,Y 282.945,Z 377.568,A -85,B 0,C 180,E1 12751.333,E2 12751.333} C_VEL
LIN {X 0,Y 289.194,Z 385.686,A -85,B 0,C 180,E1 12748.412,E2 12748.412} C_VEL
LIN {X 0,Y 296.958,Z 396.688,A -85,B 0,C 180,E1 12745.251,E2 12745.251} C_VEL
LIN {X 0,Y 305.116,Z 409.234,A -85,B 0,C 180,E1 12742.326,E2 12742.326} C_VEL
LIN {X 0,Y 313.511,Z 423.635,A -85,B 0,C 180,E1 12739.623,E2 12739.623} C_VEL
LIN {X 0,Y 315.646,Z 427.98,A -85,B 0,C 180,E1 12738.962,E2 12738.962} C_VEL
LIN {X 0,Y 307.654,Z 572.466,A -85,B 0,C 180,E1 12735.861,E2 12735.861} C_VEL
LIN {X 0,Y 306.034,Z 592.378,A -85,B 0,C 180,E1 12735.15,E2 12735.15} C_VEL
LIN {X 0,Y 303.473,Z 611.223,A -85,B 0,C 180,E1 12734.172,E2 12734.172} C_VEL
LIN {X 0,Y 299.921,Z 630.065,A -85,B 0,C 180,E1 12732.849,E2 12732.849} C_VEL
LIN {X 0,Y 295.686,Z 647.616,A -85,B 0,C 180,E1 12731.252,E2 12731.252} C_VEL
LIN {X 0,Y 290.843,Z 664.176,A -85,B 0,C 180,E1 12729.352,E2 12729.352} C_VEL
LIN {X 0,Y 285.626,Z 679.555,A -85,B 0,C 180,E1 12727.145,E2 12727.145} C_VEL
LIN {X 0,Y 280.092,Z 693.944,A -85,B 0,C 180,E1 12724.581,E2 12724.581} C_VEL
LIN {X 0,Y 274.476,Z 707.191,A -85,B 0,C 180,E1 12721.638,E2 12721.638} C_VEL
LIN {X 0,Y 269.11,Z 718.867,A -85,B 0,C 180,E1 12718.396,E2 12718.396} C_VEL
LIN {X 0,Y 264.194,Z 729.029,A -85,B 0,C 180,E1 12714.839,E2 12714.839} C_VEL
LIN {X 0,Y 259.891,Z 737.68,A -85,B 0,C 180,E1 12710.964,E2 12710.964} C_VEL
LIN {X 0,Y 256.336,Z 744.792,A -85,B 0,C 180,E1 12706.776,E2 12706.776} C_VEL
LIN {X 0,Y 253.686,Z 750.293,A -85,B 0,C 180,E1 12702.288,E2 12702.288} C_VEL
LIN {X 0,Y 252.003,Z 753.954,A -85,B 0,C 180,E1 12697.753,E2 12697.753} C_VEL
LIN {X 0,Y 251.171,Z 755.913,A -85,B 0,C 180,E1 12693.195,E2 12693.195} C_VEL
LIN {X 0,Y 251.039,Z 756.254,A -85,B 0,C 180,E1 12688.631,E2 12688.631} C_VEL
LIN {X 0,Y 251.564,Z 754.995,A -85,B 0,C 180,E1 12684.069,E2 12684.069} C_VEL
LIN {X 0,Y 252.876,Z 752.076,A -85,B 0,C 180,E1 12679.521,E2 12679.521} C_VEL
LIN {X 0,Y 255.102,Z 747.382,A -85,B 0,C 180,E1 12675.009,E2 12675.009} C_VEL
LIN {X 0,Y 258.204,Z 741.123,A -85,B 0,C 180,E1 12670.783,E2 12670.783} C_VEL
LIN {X 0,Y 262.173,Z 733.239,A -85,B 0,C 180,E1 12666.798,E2 12666.798} C_VEL
LIN {X 0,Y 266.893,Z 723.638,A -85,B 0,C 180,E1 12663.045,E2 12663.045} C_VEL
LIN {X 0,Y 271.94,Z 712.971,A -85,B 0,C 180,E1 12659.755,E2 12659.755} C_VEL
LIN {X 0,Y 277.289,Z 700.908,A -85,B 0,C 180,E1 12656.765,E2 12656.765} C_VEL
LIN {X 0,Y 282.99,Z 686.848,A -85,B 0,C 180,E1 12653.966,E2 12653.966} C_VEL
LIN {X 0,Y 288.434,Z 671.864,A -85,B 0,C 180,E1 12651.577,E2 12651.577} C_VEL
LIN {X 0,Y 293.469,Z 655.921,A -85,B 0,C 180,E1 12649.532,E2 12649.532} C_VEL
LIN {X 0,Y 298.059,Z 638.753,A -85,B 0,C 180,E1 12647.781,E2 12647.781} C_VEL
LIN {X 0,Y 301.939,Z 620.702,A -85,B 0,C 180,E1 12646.337,E2 12646.337} C_VEL
LIN {X 0,Y 305.048,Z 601.447,A -85,B 0,C 180,E1 12645.171,E2 12645.171} C_VEL
LIN {X 0,Y 307.146,Z 581.799,A -85,B 0,C 180,E1 12644.321,E2 12644.321} C_VEL
LIN {X 0,Y 308.502,Z 557.357,A -85,B 0,C 180,E1 12643.657,E2 12643.657} C_VEL
LIN {X 0,Y 315.722,Z 428.972,A -85,B 0,C 180,E1 12640.948,E2 12640.948} C_VEL
LIN {X 0,Y 315.453,Z 426.101,A -85,B 0,C 180,E1 12640.784,E2 12640.784} C_VEL
LIN {X 0,Y 314.164,Z 422.942,A -85,B 0,C 180,E1 12640.365,E2 12640.365} C_VEL
LIN {X 0,Y 311.128,Z 419.574,A -85,B 0,C 180,E1 12639.498,E2 12639.498} C_VEL
LIN {X 0,Y 301.539,Z 414.029,A -85,B 0,C 180,E1 12636.707,E2 12636.707} C_VEL
LIN {X 0,Y 299.386,Z 411.597,A -85,B 0,C 180,E1 12635.977,E2 12635.977} C_VEL
LIN {X 0,Y 291.54,Z 399.548,A -85,B 0,C 180,E1 12632.929,E2 12632.929} C_VEL
LIN {X 0,Y 283.395,Z 388.069,A -85,B 0,C 180,E1 12629.252,E2 12629.252} C_VEL
LIN {X 0,Y 278.605,Z 382.043,A -85,B 0,C 180,E1 12626.77,E2 12626.77} C_VEL
LIN {X 0,Y 274.918,Z 377.366,A -85,B 0,C 180,E1 12624.604,E2 12624.604} C_VEL
LIN {X 0,Y 270.738,Z 372.222,A -85,B 0,C 180,E1 12621.787,E2 12621.787} C_VEL
LIN {X 0,Y 266.769,Z 367.583,A -85,B 0,C 180,E1 12618.578,E2 12618.578} C_VEL
LIN {X 0,Y 260.852,Z 361.011,A -85,B 0,C 180,E1 12611.498,E2 12611.498} C_VEL
LIN {X 0,Y 259.657,Z 359.856,A -85,B 0,C 180,E1 12605.525,E2 12605.525} C_VEL
LIN {X 0,Y 260.201,Z 360.429,A -85,B 0,C 180,E1 12600,E2 12600} C_VEL
LIN {X 0,Y 261.322,Z 361.624,A -85,B 0,C 180,E1 12596.491,E2 12596.491} C_VEL
LIN {X 0,Y 264.546,Z 367.06,A -85,B 0,C 180,E1 12590.098,E2 12590.098} C_VEL
LIN {X 0,Y 268.091,Z 371.757,A -85,B 0,C 180,E1 12586.751,E2 12586.751} C_VEL
LIN {X 0,Y 273.021,Z 378.307,A -85,B 0,C 180,E1 12583.074,E2 12583.074} C_VEL
LIN {X 0,Y 277.486,Z 384.308,A -85,B 0,C 180,E1 12580.312,E2 12580.312} C_VEL
LIN {X 0,Y 283.769,Z 393.268,A -85,B 0,C 180,E1 12576.977,E2 12576.977} C_VEL
LIN {X 0,Y 289.947,Z 402.565,A -85,B 0,C 180,E1 12574.137,E2 12574.137} C_VEL
LIN {X 0,Y 297.098,Z 414.031,A -85,B 0,C 180,E1 12571.233,E2 12571.233} C_VEL
LIN {X 0,Y 305.535,Z 428.951,A -85,B 0,C 180,E1 12568.179,E2 12568.179} C_VEL
LIN {X 0,Y 311.41,Z 440.745,A -85,B 0,C 180,E1 12566.205,E2 12566.205} C_VEL
LIN {X 0,Y 299.939,Z 613.756,A -85,B 0,C 180,E1 12562.177,E2 12562.177} C_VEL
LIN {X 0,Y 297.737,Z 634.349,A -85,B 0,C 180,E1 12561.537,E2 12561.537} C_VEL
LIN {X 0,Y 294.375,Z 654.325,A -85,B 0,C 180,E1 12560.673,E2 12560.673} C_VEL
LIN {X 0,Y 289.873,Z 674.284,A -85,B 0,C 180,E1 12559.512,E2 12559.512} C_VEL
LIN {X 0,Y 284.573,Z 693.791,A -85,B 0,C 180,E1 12557.995,E2 12557.995} C_VEL
LIN {X 0,Y 278.62,Z 712.855,A -85,B 0,C 180,E1 12556.067,E2 12556.067} C_VEL
LIN {X 0,Y 272.428,Z 730.666,A -85,B 0,C 180,E1 12553.773,E2 12553.773} C_VEL
LIN {X 0,Y 266.189,Z 747.277,A -85,B 0,C 180,E1 12551.095,E2 12551.095} C_VEL
LIN {X 0,Y 260.188,Z 762.629,A -85,B 0,C 180,E1 12548.022,E2 12548.022} C_VEL
LIN {X 0,Y 254.823,Z 776.222,A -85,B 0,C 180,E1 12544.675,E2 12544.675} C_VEL
LIN {X 0,Y 249.934,Z 789.048,A -85,B 0,C 180,E1 12540.8,E2 12540.8} C_VEL
LIN {X 0,Y 245.999,Z 800.41,A -85,B 0,C 180,E1 12536.556,E2 12536.556} C_VEL
LIN {X 0,Y 243.195,Z 810.243,A -85,B 0,C 180,E1 12531.97,E2 12531.97} C_VEL
LIN {X 0,Y 241.661,Z 818.097,A -85,B 0,C 180,E1 12527.331,E2 12527.331} C_VEL
LIN {X 0,Y 241.215,Z 824.117,A -85,B 0,C 180,E1 12522.69,E2 12522.69} C_VEL
LIN {X 0,Y 241.538,Z 828.112,A -85,B 0,C 180,E1 12518.33,E2 12518.33} C_VEL
LIN {X 0,Y 242.114,Z 830.426,A -85,B 0,C 180,E1 12514.263,E2 12514.263} C_VEL
LIN {X 0,Y 242.425,Z 831.259,A -85,B 0,C 180,E1 12510.709,E2 12510.709} C_VEL
LIN {X 0,Y 242.269,Z 830.908,A -85,B 0,C 180,E1 12507.123,E2 12507.123} C_VEL
LIN {X 0,Y 241.766,Z 829.214,A -85,B 0,C 180,E1 12503.35,E2 12503.35} C_VEL
LIN {X 0,Y 241.279,Z 825.816,A -85,B 0,C 180,E1 12499.011,E2 12499.011} C_VEL
LIN {X 0,Y 241.392,Z 820.517,A -85,B 0,C 180,E1 12494.382,E2 12494.382} C_VEL
LIN {X 0,Y 242.576,Z 812.939,A -85,B 0,C 180,E1 12489.491,E2 12489.491} C_VEL
LIN {X 0,Y 244.961,Z 803.735,A -85,B 0,C 180,E1 12484.882,E2 12484.882} C_VEL
LIN {X 0,Y 248.487,Z 793.032,A -85,B 0,C 180,E1 12480.601,E2 12480.601} C_VEL
LIN {X 0,Y 252.959,Z 780.921,A -85,B 0,C 180,E1 12476.674,E2 12476.674} C_VEL
LIN {X 0,Y 258.222,Z 767.453,A -85,B 0,C 180,E1 12473.119,E2 12473.119} C_VEL
LIN {X 0,Y 264.176,Z 752.263,A -85,B 0,C 180,E1 12469.865,E2 12469.865} C_VEL
LIN {X 0,Y 270.488,Z 735.645,A -85,B 0,C 180,E1 12467.001,E2 12467.001} C_VEL
LIN {X 0,Y 276.674,Z 718.278,A -85,B 0,C 180,E1 12464.61,E2 12464.61} C_VEL
LIN {X 0,Y 282.584,Z 700.006,A -85,B 0,C 180,E1 12462.613,E2 12462.613} C_VEL
LIN {X 0,Y 287.937,Z 681.319,A -85,B 0,C 180,E1 12461.018,E2 12461.018} C_VEL
LIN {X 0,Y 292.634,Z 662.062,A -85,B 0,C 180,E1 12459.758,E2 12459.758} C_VEL
LIN {X 0,Y 296.561,Z 641.568,A -85,B 0,C 180,E1 12458.763,E2 12458.763} C_VEL
LIN {X 0,Y 299.288,Z 620.33,A -85,B 0,C 180,E1 12458.017,E2 12458.017} C_VEL
LIN {X 0,Y 311.297,Z 441.152,A -85,B 0,C 180,E1 12453.832,E2 12453.832} C_VEL
LIN {X 0,Y 310.816,Z 439.448,A -85,B 0,C 180,E1 12453.649,E2 12453.649} C_VEL
LIN {X 0,Y 302.479,Z 423.487,A -85,B 0,C 180,E1 12450.821,E2 12450.821} C_VEL
LIN {X 0,Y 294.957,Z 410.543,A -85,B 0,C 180,E1 12448.001,E2 12448.001} C_VEL
LIN {X 0,Y 287.632,Z 398.981,A -85,B 0,C 180,E1 12444.928,E2 12444.928} C_VEL
LIN {X 0,Y 281.321,Z 389.864,A -85,B 0,C 180,E1 12441.912,E2 12441.912} C_VEL
LIN {X 0,Y 275.621,Z 381.795,A -85,B 0,C 180,E1 12438.726,E2 12438.726} C_VEL
LIN {X 0,Y 271.339,Z 376.126,A -85,B 0,C 180,E1 12435.933,E2 12435.933} C_VEL
LIN {X 0,Y 267.869,Z 371.581,A -85,B 0,C 180,E1 12433.271,E2 12433.271} C_VEL
LIN {X 0,Y 264.423,Z 366.898,A -85,B 0,C 180,E1 12430.016,E2 12430.016} C_VEL
LIN {X 0,Y 261.036,Z 361.164,A -85,B 0,C 180,E1 12423.073,E2 12423.073} C_VEL
LIN {X 0,Y 259.523,Z 359.666,A -85,B 0,C 180,E1 12416.687,E2 12416.687} C_VEL
LIN {X 0,Y 259.871,Z 360.112,A -85,B 0,C 180,E1 12410.923,E2 12410.923} C_VEL
LIN {X 0,Y 261.203,Z 361.397,A -85,B 0,C 180,E1 12407.397,E2 12407.397} C_VEL
LIN {X 0,Y 265.33,Z 366.168,A -85,B 0,C 180,E1 12402.433,E2 12402.433} C_VEL
LIN {X 0,Y 266.687,Z 367.503,A -85,B 0,C 180,E1 12401.19,E2 12401.19} C_VEL
LIN {X 0,Y 270.552,Z 372.073,A -85,B 0,C 180,E1 12398.083,E2 12398.083} C_VEL
LIN {X 0,Y 271.984,Z 373.859,A -85,B 0,C 180,E1 12397.065,E2 12397.065} C_VEL
LIN {X 0,Y 276.235,Z 379.016,A -85,B 0,C 180,E1 12394.371,E2 12394.371} C_VEL
LIN {X 0,Y 280.703,Z 384.74,A -85,B 0,C 180,E1 12391.896,E2 12391.896} C_VEL
LIN {X 0,Y 286.718,Z 392.744,A -85,B 0,C 180,E1 12388.986,E2 12388.986} C_VEL
LIN {X 0,Y 294.761,Z 404.38,A -85,B 0,C 180,E1 12385.612,E2 12385.612} C_VEL
LIN {X 0,Y 303.115,Z 417.764,A -85,B 0,C 180,E1 12382.541,E2 12382.541} C_VEL
LIN {X 0,Y 310.604,Z 431.188,A -85,B 0,C 180,E1 12380.064,E2 12380.064} C_VEL
LIN {X 0,Y 302.407,Z 573.246,A -85,B 0,C 180,E1 12376.987,E2 12376.987} C_VEL
LIN {X 0,Y 300.706,Z 593.258,A -85,B 0,C 180,E1 12376.265,E2 12376.265} C_VEL
LIN {X 0,Y 298.016,Z 612.277,A -85,B 0,C 180,E1 12375.268,E2 12375.268} C_VEL
LIN {X 0,Y 294.452,Z 630.537,A -85,B 0,C 180,E1 12373.979,E2 12373.979} C_VEL
LIN {X 0,Y 290.057,Z 648.192,A -85,B 0,C 180,E1 12372.368,E2 12372.368} C_VEL
LIN {X 0,Y 284.883,Z 665.271,A -85,B 0,C 180,E1 12370.393,E2 12370.393} C_VEL
LIN {X 0,Y 279.376,Z 680.87,A -85,B 0,C 180,E1 12368.122,E2 12368.122} C_VEL
LIN {X 0,Y 273.622,Z 695.221,A -85,B 0,C 180,E1 12365.521,E2 12365.521} C_VEL
LIN {X 0,Y 267.772,Z 708.444,A -85,B 0,C 180,E1 12362.526,E2 12362.526} C_VEL
LIN {X 0,Y 262.169,Z 720.104,A -85,B 0,C 180,E1 12359.219,E2 12359.219} C_VEL
LIN {X 0,Y 257.021,Z 730.255,A -85,B 0,C 180,E1 12355.582,E2 12355.582} C_VEL
LIN {X 0,Y 252.501,Z 738.898,A -85,B 0,C 180,E1 12351.608,E2 12351.608} C_VEL
LIN {X 0,Y 248.751,Z 746.004,A -85,B 0,C 180,E1 12347.304,E2 12347.304} C_VEL
LIN {X 0,Y 245.944,Z 751.501,A -85,B 0,C 180,E1 12342.681,E2 12342.681} C_VEL
LIN {X 0,Y 244.158,Z 755.158,A -85,B 0,C 180,E1 12338.003,E2 12338.003} C_VEL
LIN {X 0,Y 243.272,Z 757.115,A -85,B 0,C 180,E1 12333.299,E2 12333.299} C_VEL
LIN {X 0,Y 243.132,Z 757.455,A -85,B 0,C 180,E1 12328.586,E2 12328.586} C_VEL
LIN {X 0,Y 243.691,Z 756.197,A -85,B 0,C 180,E1 12323.876,E2 12323.876} C_VEL
LIN {X 0,Y 245.087,Z 753.28,A -85,B 0,C 180,E1 12319.184,E2 12319.184} C_VEL
LIN {X 0,Y 247.447,Z 748.588,A -85,B 0,C 180,E1 12314.533,E2 12314.533} C_VEL
LIN {X 0,Y 250.725,Z 742.333,A -85,B 0,C 180,E1 12310.187,E2 12310.187} C_VEL
LIN {X 0,Y 255.002,Z 734.264,A -85,B 0,C 180,E1 12306.008,E2 12306.008} C_VEL
LIN {X 0,Y 259.856,Z 724.856,A -85,B 0,C 180,E1 12302.25,E2 12302.25} C_VEL
LIN {X 0,Y 265.196,Z 714.075,A -85,B 0,C 180,E1 12298.855,E2 12298.855} C_VEL
LIN {X 0,Y 270.812,Z 701.935,A -85,B 0,C 180,E1 12295.795,E2 12295.795} C_VEL
LIN {X 0,Y 276.596,Z 688.252,A -85,B 0,C 180,E1 12293.025,E2 12293.025} C_VEL
LIN {X 0,Y 282.168,Z 673.561,A -85,B 0,C 180,E1 12290.634,E2 12290.634} C_VEL
LIN {X 0,Y 287.521,Z 657.318,A -85,B 0,C 180,E1 12288.513,E2 12288.513} C_VEL
LIN {X 0,Y 292.369,Z 639.895,A -85,B 0,C 180,E1 12286.712,E2 12286.712} C_VEL
LIN {X 0,Y 296.306,Z 622.353,A -85,B 0,C 180,E1 12285.288,E2 12285.288} C_VEL
LIN {X 0,Y 299.493,Z 603.691,A -85,B 0,C 180,E1 12284.131,E2 12284.131} C_VEL
LIN {X 0,Y 301.707,Z 584.601,A -85,B 0,C 180,E1 12283.27,E2 12283.27} C_VEL
LIN {X 0,Y 303.053,Z 563.144,A -85,B 0,C 180,E1 12282.641,E2 12282.641} C_VEL
LIN {X 0,Y 310.65,Z 431.116,A -85,B 0,C 180,E1 12279.8,E2 12279.8} C_VEL
LIN {X 0,Y 302.651,Z 416.894,A -85,B 0,C 180,E1 12277.139,E2 12277.139} C_VEL
LIN {X 0,Y 299.386,Z 411.597,A -85,B 0,C 180,E1 12275.977,E2 12275.977} C_VEL
LIN {X 0,Y 296.103,Z 407.988,A -85,B 0,C 180,E1 12274.815,E2 12274.815} C_VEL
LIN {X 0,Y 288.445,Z 403.385,A -85,B 0,C 180,E1 12272.017,E2 12272.017} C_VEL
LIN {X 0,Y 284.803,Z 400.362,A -85,B 0,C 180,E1 12270.49,E2 12270.49} C_VEL
LIN {X 0,Y 284.011,Z 399.335,A -85,B 0,C 180,E1 12270.122,E2 12270.122} C_VEL
LIN {X 0,Y 277.331,Z 390.187,A -85,B 0,C 180,E1 12266.671,E2 12266.671} C_VEL
LIN {X 0,Y 273.037,Z 384.773,A -85,B 0,C 180,E1 12264.099,E2 12264.099} C_VEL
LIN {X 0,Y 268.964,Z 379.69,A -85,B 0,C 180,E1 12261.251,E2 12261.251} C_VEL
LIN {X 0,Y 264.482,Z 374.303,A -85,B 0,C 180,E1 12257.377,E2 12257.377} C_VEL
LIN {X 0,Y 259.636,Z 368.814,A -85,B 0,C 180,E1 12251.102,E2 12251.102} C_VEL
LIN {X 0,Y 257.497,Z 367.549,A -85,B 0,C 180,E1 12244.901,E2 12244.901} C_VEL
LIN {X 0,Y 258.026,Z 368.268,A -85,B 0,C 180,E1 12239.112,E2 12239.112} C_VEL
LIN {X 0,Y 259.052,Z 369.438,A -85,B 0,C 180,E1 12236.46,E2 12236.46} C_VEL
LIN {X 0,Y 263.131,Z 374.76,A -85,B 0,C 180,E1 12230.486,E2 12230.486} C_VEL
LIN {X 0,Y 266.716,Z 379.556,A -85,B 0,C 180,E1 12227.002,E2 12227.002} C_VEL
LIN {X 0,Y 271.243,Z 385.883,A -85,B 0,C 180,E1 12223.511,E2 12223.511} C_VEL
LIN {X 0,Y 275.28,Z 391.416,A -85,B 0,C 180,E1 12220.92,E2 12220.92} C_VEL
LIN {X 0,Y 281.392,Z 400.399,A -85,B 0,C 180,E1 12217.544,E2 12217.544} C_VEL
LIN {X 0,Y 287.329,Z 409.57,A -85,B 0,C 180,E1 12214.714,E2 12214.714} C_VEL
LIN {X 0,Y 294.659,Z 421.67,A -85,B 0,C 180,E1 12211.637,E2 12211.637} C_VEL
LIN {X 0,Y 302.459,Z 436.06,A -85,B 0,C 180,E1 12208.707,E2 12208.707} C_VEL
LIN {X 0,Y 306.465,Z 444.425,A -85,B 0,C 180,E1 12207.295,E2 12207.295} C_VEL
LIN {X 0,Y 294.167,Z 620.486,A -85,B 0,C 180,E1 12203.171,E2 12203.171} C_VEL
LIN {X 0,Y 291.22,Z 642.131,A -85,B 0,C 180,E1 12202.393,E2 12202.393} C_VEL
LIN {X 0,Y 287.038,Z 662.887,A -85,B 0,C 180,E1 12201.363,E2 12201.363} C_VEL
LIN {X 0,Y 281.883,Z 682.993,A -85,B 0,C 180,E1 12200.009,E2 12200.009} C_VEL
LIN {X 0,Y 275.966,Z 702.468,A -85,B 0,C 180,E1 12198.274,E2 12198.274} C_VEL
LIN {X 0,Y 269.637,Z 720.875,A -85,B 0,C 180,E1 12196.155,E2 12196.155} C_VEL
LIN {X 0,Y 263.056,Z 738.26,A -85,B 0,C 180,E1 12193.618,E2 12193.618} C_VEL
LIN {X 0,Y 256.451,Z 754.612,A -85,B 0,C 180,E1 12190.624,E2 12190.624} C_VEL
LIN {X 0,Y 250.498,Z 768.957,A -85,B 0,C 180,E1 12187.35,E2 12187.35} C_VEL
LIN {X 0,Y 245.055,Z 782.1,A -85,B 0,C 180,E1 12183.66,E2 12183.66} C_VEL
LIN {X 0,Y 240.296,Z 794.336,A -85,B 0,C 180,E1 12179.405,E2 12179.405} C_VEL
LIN {X 0,Y 236.778,Z 804.563,A -85,B 0,C 180,E1 12174.978,E2 12174.978} C_VEL
LIN {X 0,Y 234.442,Z 813.342,A -85,B 0,C 180,E1 12170.209,E2 12170.209} C_VEL
LIN {X 0,Y 233.388,Z 820.231,A -85,B 0,C 180,E1 12165.403,E2 12165.403} C_VEL
LIN {X 0,Y 233.343,Z 825.326,A -85,B 0,C 180,E1 12160.617,E2 12160.617} C_VEL
LIN {X 0,Y 233.866,Z 828.29,A -85,B 0,C 180,E1 12156.382,E2 12156.382} C_VEL
LIN {X 0,Y 234.393,Z 829.845,A -85,B 0,C 180,E1 12152.445,E2 12152.445} C_VEL
LIN {X 0,Y 234.505,Z 830.027,A -85,B 0,C 180,E1 12149.023,E2 12149.023} C_VEL
LIN {X 0,Y 234.129,Z 829.119,A -85,B 0,C 180,E1 12145.346,E2 12145.346} C_VEL
LIN {X 0,Y 233.501,Z 826.48,A -85,B 0,C 180,E1 12140.884,E2 12140.884} C_VEL
LIN {X 0,Y 233.278,Z 821.992,A -85,B 0,C 180,E1 12136.112,E2 12136.112} C_VEL
LIN {X 0,Y 233.979,Z 815.722,A -85,B 0,C 180,E1 12131.308,E2 12131.308} C_VEL
LIN {X 0,Y 235.899,Z 807.55,A -85,B 0,C 180,E1 12126.521,E2 12126.521} C_VEL
LIN {X 0,Y 239.182,Z 797.347,A -85,B 0,C 180,E1 12121.812,E2 12121.812} C_VEL
LIN {X 0,Y 243.627,Z 785.587,A -85,B 0,C 180,E1 12117.478,E2 12117.478} C_VEL
LIN {X 0,Y 248.697,Z 773.145,A -85,B 0,C 180,E1 12113.773,E2 12113.773} C_VEL
LIN {X 0,Y 254.544,Z 759.011,A -85,B 0,C 180,E1 12110.344,E2 12110.344} C_VEL
LIN {X 0,Y 260.913,Z 743.411,A -85,B 0,C 180,E1 12107.291,E2 12107.291} C_VEL
LIN {X 0,Y 267.509,Z 726.344,A -85,B 0,C 180,E1 12104.617,E2 12104.617} C_VEL
LIN {X 0,Y 273.686,Z 708.928,A -85,B 0,C 180,E1 12102.443,E2 12102.443} C_VEL
LIN {X 0,Y 279.444,Z 690.889,A -85,B 0,C 180,E1 12100.666,E2 12100.666} C_VEL
LIN {X 0,Y 284.678,Z 672.092,A -85,B 0,C 180,E1 12099.231,E2 12099.231} C_VEL
LIN {X 0,Y 289.362,Z 651.581,A -85,B 0,C 180,E1 12098.059,E2 12098.059} C_VEL
LIN {X 0,Y 292.884,Z 630.334,A -85,B 0,C 180,E1 12097.17,E2 12097.17} C_VEL
LIN {X 0,Y 295.042,Z 608.532,A -85,B 0,C 180,E1 12096.533,E2 12096.533} C_VEL
LIN {X 0,Y 306.312,Z 443.938,A -85,B 0,C 180,E1 12092.698,E2 12092.698} C_VEL
LIN {X 0,Y 298.667,Z 429.025,A -85,B 0,C 180,E1 12089.976,E2 12089.976} C_VEL
LIN {X 0,Y 291.575,Z 416.554,A -85,B 0,C 180,E1 12087.189,E2 12087.189} C_VEL
LIN {X 0,Y 284.887,Z 405.688,A -85,B 0,C 180,E1 12084.244,E2 12084.244} C_VEL
LIN {X 0,Y 278.845,Z 396.729,A -85,B 0,C 180,E1 12081.232,E2 12081.232} C_VEL
LIN {X 0,Y 273.307,Z 388.764,A -85,B 0,C 180,E1 12078.006,E2 12078.006} C_VEL
LIN {X 0,Y 269.459,Z 383.477,A -85,B 0,C 180,E1 12075.385,E2 12075.385} C_VEL
LIN {X 0,Y 266.219,Z 379.13,A -85,B 0,C 180,E1 12072.802,E2 12072.802} C_VEL
LIN {X 0,Y 262.412,Z 373.892,A -85,B 0,C 180,E1 12068.987,E2 12068.987} C_VEL
LIN {X 0,Y 258.498,Z 368.712,A -85,B 0,C 180,E1 12062.882,E2 12062.882} C_VEL
LIN {X 0,Y 257.124,Z 367.282,A -85,B 0,C 180,E1 12056.432,E2 12056.432} C_VEL
LIN {X 0,Y 258.634,Z 368.161,A -85,B 0,C 180,E1 12050.206,E2 12050.206} C_VEL
LIN {X 0,Y 260.244,Z 369.538,A -85,B 0,C 180,E1 12047.35,E2 12047.35} C_VEL
LIN {X 0,Y 264.157,Z 374.05,A -85,B 0,C 180,E1 12042.601,E2 12042.601} C_VEL
LIN {X 0,Y 265.383,Z 375.444,A -85,B 0,C 180,E1 12041.436,E2 12041.436} C_VEL
LIN {X 0,Y 269.346,Z 380.009,A -85,B 0,C 180,E1 12038.209,E2 12038.209} C_VEL
LIN {X 0,Y 274.462,Z 386.667,A -85,B 0,C 180,E1 12034.771,E2 12034.771} C_VEL
LIN {X 0,Y 278.575,Z 392.041,A -85,B 0,C 180,E1 12032.418,E2 12032.418} C_VEL
LIN {X 0,Y 284.268,Z 399.8,A -85,B 0,C 180,E1 12029.569,E2 12029.569} C_VEL
LIN {X 0,Y 291.804,Z 410.986,A -85,B 0,C 180,E1 12026.283,E2 12026.283} C_VEL
LIN {X 0,Y 299.681,Z 423.896,A -85,B 0,C 180,E1 12023.269,E2 12023.269} C_VEL
LIN {X 0,Y 305.653,Z 435.016,A -85,B 0,C 180,E1 12021.187,E2 12021.187} C_VEL
LIN {X 0,Y 297.3,Z 573.705,A -85,B 0,C 180,E1 12018.161,E2 12018.161} C_VEL
LIN {X 0,Y 295.55,Z 593.68,A -85,B 0,C 180,E1 12017.44,E2 12017.44} C_VEL
LIN {X 0,Y 292.801,Z 612.599,A -85,B 0,C 180,E1 12016.45,E2 12016.45} C_VEL
LIN {X 0,Y 289.102,Z 631.006,A -85,B 0,C 180,E1 12015.151,E2 12015.151} C_VEL
LIN {X 0,Y 284.543,Z 648.768,A -85,B 0,C 180,E1 12013.528,E2 12013.528} C_VEL
LIN {X 0,Y 279.319,Z 665.496,A -85,B 0,C 180,E1 12011.592,E2 12011.592} C_VEL
LIN {X 0,Y 273.668,Z 681.017,A -85,B 0,C 180,E1 12009.336,E2 12009.336} C_VEL
LIN {X 0,Y 267.659,Z 695.529,A -85,B 0,C 180,E1 12006.703,E2 12006.703} C_VEL
LIN {X 0,Y 261.523,Z 708.893,A -85,B 0,C 180,E1 12003.666,E2 12003.666} C_VEL
LIN {X 0,Y 255.629,Z 720.676,A -85,B 0,C 180,E1 12000.302,E2 12000.302} C_VEL
LIN {X 0,Y 250.186,Z 730.94,A -85,B 0,C 180,E1 11996.589,E2 11996.589} C_VEL
LIN {X 0,Y 245.383,Z 739.687,A -85,B 0,C 180,E1 11992.52,E2 11992.52} C_VEL
LIN {X 0,Y 241.368,Z 746.89,A -85,B 0,C 180,E1 11988.1,E2 11988.1} C_VEL
LIN {X 0,Y 238.336,Z 752.477,A -85,B 0,C 180,E1 11983.34,E2 11983.34} C_VEL
LIN {X 0,Y 236.388,Z 756.219,A -85,B 0,C 180,E1 11978.513,E2 11978.513} C_VEL
LIN {X 0,Y 235.4,Z 758.256,A -85,B 0,C 180,E1 11973.653,E2 11973.653} C_VEL
LIN {X 0,Y 235.216,Z 758.676,A -85,B 0,C 180,E1 11968.782,E2 11968.782} C_VEL
LIN {X 0,Y 235.771,Z 757.501,A -85,B 0,C 180,E1 11963.914,E2 11963.914} C_VEL
LIN {X 0,Y 237.208,Z 754.67,A -85,B 0,C 180,E1 11959.066,E2 11959.066} C_VEL
LIN {X 0,Y 239.658,Z 750.072,A -85,B 0,C 180,E1 11954.266,E2 11954.266} C_VEL
LIN {X 0,Y 243.275,Z 743.544,A -85,B 0,C 180,E1 11949.553,E2 11949.553} C_VEL
LIN {X 0,Y 247.587,Z 735.82,A -85,B 0,C 180,E1 11945.421,E2 11945.421} C_VEL
LIN {X 0,Y 252.864,Z 726.09,A -85,B 0,C 180,E1 11941.417,E2 11941.417} C_VEL
LIN {X 0,Y 258.607,Z 715.007,A -85,B 0,C 180,E1 11937.858,E2 11937.858} C_VEL
LIN {X 0,Y 264.609,Z 702.544,A -85,B 0,C 180,E1 11934.682,E2 11934.682} C_VEL
LIN {X 0,Y 270.597,Z 688.893,A -85,B 0,C 180,E1 11931.899,E2 11931.899} C_VEL
LIN {X 0,Y 276.586,Z 673.604,A -85,B 0,C 180,E1 11929.407,E2 11929.407} C_VEL
LIN {X 0,Y 282.163,Z 657.139,A -85,B 0,C 180,E1 11927.268,E2 11927.268} C_VEL
LIN {X 0,Y 286.946,Z 640.408,A -85,B 0,C 180,E1 11925.544,E2 11925.544} C_VEL
LIN {X 0,Y 291.03,Z 622.739,A -85,B 0,C 180,E1 11924.109,E2 11924.109} C_VEL
LIN {X 0,Y 294.382,Z 603.565,A -85,B 0,C 180,E1 11922.926,E2 11922.926} C_VEL
LIN {X 0,Y 296.689,Z 583.8,A -85,B 0,C 180,E1 11922.051,E2 11922.051} C_VEL
LIN {X 0,Y 298.203,Z 559.266,A -85,B 0,C 180,E1 11921.365,E2 11921.365} C_VEL
LIN {X 0,Y 305.696,Z 434.6,A -85,B 0,C 180,E1 11918.662,E2 11918.662} C_VEL
LIN {X 0,Y 297.082,Z 419.319,A -85,B 0,C 180,E1 11915.609,E2 11915.609} C_VEL
LIN {X 0,Y 288.785,Z 406.306,A -85,B 0,C 180,E1 11912.281,E2 11912.281} C_VEL
LIN {X 0,Y 284.011,Z 399.335,A -85,B 0,C 180,E1 11910.122,E2 11910.122} C_VEL
LIN {X 0,Y 281.149,Z 396.523,A -85,B 0,C 180,E1 11908.78,E2 11908.78} C_VEL
LIN {X 0,Y 276.362,Z 394.63,A -85,B 0,C 180,E1 11906.484,E2 11906.484} C_VEL
LIN {X 0,Y 271.794,Z 392.717,A -85,B 0,C 180,E1 11903.976,E2 11903.976} C_VEL
LIN {X 0,Y 270.944,Z 391.928,A -85,B 0,C 180,E1 11903.434,E2 11903.434} C_VEL
LIN {X 0,Y 267.351,Z 387.273,A -85,B 0,C 180,E1 11900.812,E2 11900.812} C_VEL
LIN {X 0,Y 263.114,Z 382.029,A -85,B 0,C 180,E1 11897.015,E2 11897.015} C_VEL
LIN {X 0,Y 258.557,Z 376.707,A -85,B 0,C 180,E1 11890.923,E2 11890.923} C_VEL
LIN {X 0,Y 256.5,Z 375.483,A -85,B 0,C 180,E1 11884.696,E2 11884.696} C_VEL
LIN {X 0,Y 257.092,Z 376.28,A -85,B 0,C 180,E1 11878.886,E2 11878.886} C_VEL
LIN {X 0,Y 257.981,Z 377.437,A -85,B 0,C 180,E1 11876.556,E2 11876.556} C_VEL
LIN {X 0,Y 261.729,Z 382.457,A -85,B 0,C 180,E1 11870.878,E2 11870.878} C_VEL
LIN {X 0,Y 265.913,Z 388.376,A -85,B 0,C 180,E1 11866.741,E2 11866.741} C_VEL
LIN {X 0,Y 269.411,Z 393.338,A -85,B 0,C 180,E1 11864.005,E2 11864.005} C_VEL
LIN {X 0,Y 273.262,Z 398.777,A -85,B 0,C 180,E1 11861.438,E2 11861.438} C_VEL
LIN {X 0,Y 279.044,Z 407.526,A -85,B 0,C 180,E1 11858.121,E2 11858.121} C_VEL
LIN {X 0,Y 285.652,Z 417.93,A -85,B 0,C 180,E1 11854.887,E2 11854.887} C_VEL
LIN {X 0,Y 292.882,Z 430.603,A -85,B 0,C 180,E1 11851.783,E2 11851.783} C_VEL
LIN {X 0,Y 300.457,Z 445.23,A -85,B 0,C 180,E1 11848.865,E2 11848.865} C_VEL
LIN {X 0,Y 301.565,Z 447.913,A -85,B 0,C 180,E1 11848.445,E2 11848.445} C_VEL
LIN {X 0,Y 289.159,Z 619.599,A -85,B 0,C 180,E1 11844.411,E2 11844.411} C_VEL
LIN {X 0,Y 286.148,Z 641.14,A -85,B 0,C 180,E1 11843.637,E2 11843.637} C_VEL
LIN {X 0,Y 281.87,Z 661.827,A -85,B 0,C 180,E1 11842.613,E2 11842.613} C_VEL
LIN {X 0,Y 276.706,Z 681.385,A -85,B 0,C 180,E1 11841.304,E2 11841.304} C_VEL
LIN {X 0,Y 270.978,Z 699.735,A -85,B 0,C 180,E1 11839.689,E2 11839.689} C_VEL
LIN {X 0,Y 264.827,Z 717.159,A -85,B 0,C 180,E1 11837.73,E2 11837.73} C_VEL
LIN {X 0,Y 258.142,Z 734.335,A -85,B 0,C 180,E1 11835.294,E2 11835.294} C_VEL
LIN {X 0,Y 251.348,Z 750.591,A -85,B 0,C 180,E1 11832.396,E2 11832.396} C_VEL
LIN {X 0,Y 244.707,Z 765.827,A -85,B 0,C 180,E1 11828.992,E2 11828.992} C_VEL
LIN {X 0,Y 238.534,Z 779.922,A -85,B 0,C 180,E1 11825.047,E2 11825.047} C_VEL
LIN {X 0,Y 233.305,Z 792.414,A -85,B 0,C 180,E1 11820.662,E2 11820.662} C_VEL
LIN {X 0,Y 229.251,Z 803.286,A -85,B 0,C 180,E1 11815.857,E2 11815.857} C_VEL
LIN {X 0,Y 226.686,Z 812.077,A -85,B 0,C 180,E1 11810.932,E2 11810.932} C_VEL
LIN {X 0,Y 225.473,Z 818.98,A -85,B 0,C 180,E1 11805.958,E2 11805.958} C_VEL
LIN {X 0,Y 225.358,Z 824.09,A -85,B 0,C 180,E1 11800.998,E2 11800.998} C_VEL
LIN {X 0,Y 225.895,Z 827.071,A -85,B 0,C 180,E1 11796.608,E2 11796.608} C_VEL
LIN {X 0,Y 226.468,Z 828.64,A -85,B 0,C 180,E1 11792.53,E2 11792.53} C_VEL
LIN {X 0,Y 226.592,Z 828.825,A -85,B 0,C 180,E1 11788.989,E2 11788.989} C_VEL
LIN {X 0,Y 226.217,Z 827.996,A -85,B 0,C 180,E1 11785.437,E2 11785.437} C_VEL
LIN {X 0,Y 225.544,Z 825.443,A -85,B 0,C 180,E1 11780.817,E2 11780.817} C_VEL
LIN {X 0,Y 225.306,Z 821.337,A -85,B 0,C 180,E1 11776.135,E2 11776.135} C_VEL
LIN {X 0,Y 226.015,Z 815.194,A -85,B 0,C 180,E1 11771.16,E2 11771.16} C_VEL
LIN {X 0,Y 228.001,Z 807.19,A -85,B 0,C 180,E1 11766.207,E2 11766.207} C_VEL
LIN {X 0,Y 231.197,Z 797.77,A -85,B 0,C 180,E1 11761.595,E2 11761.595} C_VEL
LIN {X 0,Y 235.747,Z 786.348,A -85,B 0,C 180,E1 11757.115,E2 11757.115} C_VEL
LIN {X 0,Y 241.29,Z 773.485,A -85,B 0,C 180,E1 11753.07,E2 11753.07} C_VEL
LIN {X 0,Y 247.734,Z 758.735,A -85,B 0,C 180,E1 11749.355,E2 11749.355} C_VEL
LIN {X 0,Y 254.404,Z 743.211,A -85,B 0,C 180,E1 11746.236,E2 11746.236} C_VEL
LIN {X 0,Y 261.141,Z 726.599,A -85,B 0,C 180,E1 11743.565,E2 11743.565} C_VEL
LIN {X 0,Y 267.636,Z 709.13,A -85,B 0,C 180,E1 11741.332,E2 11741.332} C_VEL
LIN {X 0,Y 273.575,Z 691.374,A -85,B 0,C 180,E1 11739.544,E2 11739.544} C_VEL
LIN {X 0,Y 279.247,Z 671.79,A -85,B 0,C 180,E1 11738.029,E2 11738.029} C_VEL
LIN {X 0,Y 284.026,Z 651.633,A -85,B 0,C 180,E1 11736.866,E2 11736.866} C_VEL
LIN {X 0,Y 287.728,Z 630.265,A -85,B 0,C 180,E1 11735.959,E2 11735.959} C_VEL
LIN {X 0,Y 290.003,Z 608.45,A -85,B 0,C 180,E1 11735.313,E2 11735.313} C_VEL
LIN {X 0,Y 301.425,Z 447.468,A -85,B 0,C 180,E1 11731.552,E2 11731.552} C_VEL
LIN {X 0,Y 294.484,Z 433.716,A -85,B 0,C 180,E1 11728.935,E2 11728.935} C_VEL
LIN {X 0,Y 287.224,Z 420.756,A -85,B 0,C 180,E1 11725.904,E2 11725.904} C_VEL
LIN {X 0,Y 280.376,Z 409.547,A -85,B 0,C 180,E1 11722.652,E2 11722.652} C_VEL
LIN {X 0,Y 274.472,Z 400.605,A -85,B 0,C 180,E1 11719.415,E2 11719.415} C_VEL
LIN {X 0,Y 271.055,Z 395.721,A -85,B 0,C 180,E1 11717.274,E2 11717.274} C_VEL
LIN {X 0,Y 267.364,Z 390.484,A -85,B 0,C 180,E1 11714.621,E2 11714.621} C_VEL
LIN {X 0,Y 264.503,Z 386.557,A -85,B 0,C 180,E1 11712.221,E2 11712.221} C_VEL
LIN {X 0,Y 261.043,Z 381.597,A -85,B 0,C 180,E1 11708.591,E2 11708.591} C_VEL
LIN {X 0,Y 257.415,Z 376.588,A -85,B 0,C 180,E1 11702.671,E2 11702.671} C_VEL
LIN {X 0,Y 256.15,Z 375.222,A -85,B 0,C 180,E1 11696.419,E2 11696.419} C_VEL
LIN {X 0,Y 257.568,Z 376.056,A -85,B 0,C 180,E1 11690.391,E2 11690.391} C_VEL
LIN {X 0,Y 259.069,Z 377.366,A -85,B 0,C 180,E1 11687.631,E2 11687.631} C_VEL
LIN {X 0,Y 262.995,Z 381.948,A -85,B 0,C 180,E1 11682.749,E2 11682.749} C_VEL
LIN {X 0,Y 268.301,Z 388.521,A -85,B 0,C 180,E1 11678.177,E2 11678.177} C_VEL
LIN {X 0,Y 272.616,Z 394.185,A -85,B 0,C 180,E1 11675.226,E2 11675.226} C_VEL
LIN {X 0,Y 276.563,Z 399.467,A -85,B 0,C 180,E1 11672.901,E2 11672.901} C_VEL
LIN {X 0,Y 281.943,Z 406.999,A -85,B 0,C 180,E1 11670.115,E2 11670.115} C_VEL
LIN {X 0,Y 288.994,Z 417.776,A -85,B 0,C 180,E1 11666.921,E2 11666.921} C_VEL
LIN {X 0,Y 296.356,Z 430.137,A -85,B 0,C 180,E1 11663.992,E2 11663.992} C_VEL
LIN {X 0,Y 300.821,Z 438.681,A -85,B 0,C 180,E1 11662.35,E2 11662.35} C_VEL
LIN {X 0,Y 292.308,Z 574.377,A -85,B 0,C 180,E1 11659.369,E2 11659.369} C_VEL
LIN {X 0,Y 290.51,Z 594.197,A -85,B 0,C 180,E1 11658.652,E2 11658.652} C_VEL
LIN {X 0,Y 287.595,Z 613.573,A -85,B 0,C 180,E1 11657.634,E2 11657.634} C_VEL
LIN {X 0,Y 283.709,Z 632.181,A -85,B 0,C 180,E1 11656.31,E2 11656.31} C_VEL
LIN {X 0,Y 278.888,Z 650.216,A -85,B 0,C 180,E1 11654.642,E2 11654.642} C_VEL
LIN {X 0,Y 273.57,Z 666.596,A -85,B 0,C 180,E1 11652.724,E2 11652.724} C_VEL
LIN {X 0,Y 267.61,Z 682.332,A -85,B 0,C 180,E1 11650.408,E2 11650.408} C_VEL
LIN {X 0,Y 261.367,Z 696.808,A -85,B 0,C 180,E1 11647.739,E2 11647.739} C_VEL
LIN {X 0,Y 254.976,Z 710.147,A -85,B 0,C 180,E1 11644.652,E2 11644.652} C_VEL
LIN {X 0,Y 248.823,Z 721.912,A -85,B 0,C 180,E1 11641.222,E2 11641.222} C_VEL
LIN {X 0,Y 243.121,Z 732.163,A -85,B 0,C 180,E1 11637.426,E2 11637.426} C_VEL
LIN {X 0,Y 238.075,Z 740.901,A -85,B 0,C 180,E1 11633.251,E2 11633.251} C_VEL
LIN {X 0,Y 233.84,Z 748.099,A -85,B 0,C 180,E1 11628.704,E2 11628.704} C_VEL
LIN {X 0,Y 230.628,Z 753.683,A -85,B 0,C 180,E1 11623.794,E2 11623.794} C_VEL
LIN {X 0,Y 228.557,Z 757.423,A -85,B 0,C 180,E1 11618.807,E2 11618.807} C_VEL
LIN {X 0,Y 227.505,Z 759.458,A -85,B 0,C 180,E1 11613.78,E2 11613.78} C_VEL
LIN {X 0,Y 227.308,Z 759.877,A -85,B 0,C 180,E1 11608.74,E2 11608.74} C_VEL
LIN {X 0,Y 227.901,Z 758.703,A -85,B 0,C 180,E1 11603.703,E2 11603.703} C_VEL
LIN {X 0,Y 229.437,Z 755.864,A -85,B 0,C 180,E1 11598.676,E2 11598.676} C_VEL
LIN {X 0,Y 232.031,Z 751.28,A -85,B 0,C 180,E1 11593.735,E2 11593.735} C_VEL
LIN {X 0,Y 235.857,Z 744.755,A -85,B 0,C 180,E1 11588.88,E2 11588.88} C_VEL
LIN {X 0,Y 240.395,Z 737.036,A -85,B 0,C 180,E1 11584.635,E2 11584.635} C_VEL
LIN {X 0,Y 245.933,Z 727.313,A -85,B 0,C 180,E1 11580.533,E2 11580.533} C_VEL
LIN {X 0,Y 251.704,Z 716.687,A -85,B 0,C 180,E1 11577.03,E2 11577.03} C_VEL
LIN {X 0,Y 258.196,Z 703.801,A -85,B 0,C 180,E1 11573.667,E2 11573.667} C_VEL
LIN {X 0,Y 264.573,Z 689.844,A -85,B 0,C 180,E1 11570.781,E2 11570.781} C_VEL
LIN {X 0,Y 270.644,Z 674.935,A -85,B 0,C 180,E1 11568.32,E2 11568.32} C_VEL
LIN {X 0,Y 276.427,Z 658.533,A -85,B 0,C 180,E1 11566.16,E2 11566.16} C_VEL
LIN {X 0,Y 281.647,Z 640.917,A -85,B 0,C 180,E1 11564.331,E2 11564.331} C_VEL
LIN {X 0,Y 285.882,Z 623.12,A -85,B 0,C 180,E1 11562.887,E2 11562.887} C_VEL
LIN {X 0,Y 289.324,Z 603.974,A -85,B 0,C 180,E1 11561.708,E2 11561.708} C_VEL
LIN {X 0,Y 291.689,Z 584.308,A -85,B 0,C 180,E1 11560.838,E2 11560.838} C_VEL
LIN {X 0,Y 293.267,Z 559.696,A -85,B 0,C 180,E1 11560.148,E2 11560.148} C_VEL
LIN {X 0,Y 300.922,Z 438.413,A -85,B 0,C 180,E1 11557.513,E2 11557.513} C_VEL
LIN {X 0,Y 293.599,Z 425.217,A -85,B 0,C 180,E1 11554.78,E2 11554.78} C_VEL
LIN {X 0,Y 285.958,Z 412.916,A -85,B 0,C 180,E1 11551.575,E2 11551.575} C_VEL
LIN {X 0,Y 278.692,Z 402.195,A -85,B 0,C 180,E1 11548.034,E2 11548.034} C_VEL
LIN {X 0,Y 274.332,Z 396.407,A -85,B 0,C 180,E1 11545.589,E2 11545.589} C_VEL
LIN {X 0,Y 271.016,Z 392.007,A -85,B 0,C 180,E1 11543.481,E2 11543.481} C_VEL
LIN {X 0,Y 270.944,Z 391.928,A -85,B 0,C 180,E1 11543.434,E2 11543.434} C_VEL
LIN {X 0,Y 268.454,Z 390.258,A -85,B 0,C 180,E1 11541.789,E2 11541.789} C_VEL
LIN {X 0,Y 261.646,Z 389.615,A -85,B 0,C 180,E1 11536.543,E2 11536.543} C_VEL
LIN {X 0,Y 261.183,Z 389.307,A -85,B 0,C 180,E1 11536.067,E2 11536.067} C_VEL
LIN {X 0,Y 257.474,Z 384.599,A -85,B 0,C 180,E1 11530.743,E2 11530.743} C_VEL
LIN {X 0,Y 255.529,Z 383.424,A -85,B 0,C 180,E1 11524.714,E2 11524.714} C_VEL
LIN {X 0,Y 256.047,Z 384.17,A -85,B 0,C 180,E1 11519.105,E2 11519.105} C_VEL
LIN {X 0,Y 256.846,Z 385.226,A -85,B 0,C 180,E1 11516.876,E2 11516.876} C_VEL
LIN {X 0,Y 260.346,Z 390.15,A -85,B 0,C 180,E1 11511.275,E2 11511.275} C_VEL
LIN {X 0,Y 264.395,Z 396.089,A -85,B 0,C 180,E1 11507.108,E2 11507.108} C_VEL
LIN {X 0,Y 267.601,Z 400.785,A -85,B 0,C 180,E1 11504.506,E2 11504.506} C_VEL
LIN {X 0,Y 271.269,Z 406.134,A -85,B 0,C 180,E1 11501.965,E2 11501.965} C_VEL
LIN {X 0,Y 276.735,Z 414.653,A -85,B 0,C 180,E1 11498.709,E2 11498.709} C_VEL
LIN {X 0,Y 282.895,Z 424.631,A -85,B 0,C 180,E1 11495.574,E2 11495.574} C_VEL
LIN {X 0,Y 289.751,Z 437.071,A -85,B 0,C 180,E1 11492.486,E2 11492.486} C_VEL
LIN {X 0,Y 296.819,Z 451.107,A -85,B 0,C 180,E1 11489.642,E2 11489.642} C_VEL
LIN {X 0,Y 284.291,Z 618.719,A -85,B 0,C 180,E1 11485.694,E2 11485.694} C_VEL
LIN {X 0,Y 281.194,Z 640.264,A -85,B 0,C 180,E1 11484.92,E2 11484.92} C_VEL
LIN {X 0,Y 276.844,Z 660.774,A -85,B 0,C 180,E1 11483.909,E2 11483.909} C_VEL
LIN {X 0,Y 271.301,Z 681.09,A -85,B 0,C 180,E1 11482.549,E2 11482.549} C_VEL
LIN {X 0,Y 265.037,Z 700.385,A -85,B 0,C 180,E1 11480.826,E2 11480.826} C_VEL
LIN {X 0,Y 258.217,Z 718.776,A -85,B 0,C 180,E1 11478.692,E2 11478.692} C_VEL
LIN {X 0,Y 251.075,Z 736.136,A -85,B 0,C 180,E1 11476.118,E2 11476.118} C_VEL
LIN {X 0,Y 244.095,Z 751.924,A -85,B 0,C 180,E1 11473.16,E2 11473.16} C_VEL
LIN {X 0,Y 237.463,Z 766.313,A -85,B 0,C 180,E1 11469.791,E2 11469.791} C_VEL
LIN {X 0,Y 231.406,Z 779.378,A -85,B 0,C 180,E1 11465.988,E2 11465.988} C_VEL
LIN {X 0,Y 225.893,Z 791.752,A -85,B 0,C 180,E1 11461.485,E2 11461.485} C_VEL
LIN {X 0,Y 221.593,Z 802.519,A -85,B 0,C 180,E1 11456.531,E2 11456.531} C_VEL
LIN {X 0,Y 218.849,Z 811.216,A -85,B 0,C 180,E1 11451.437,E2 11451.437} C_VEL
LIN {X 0,Y 217.501,Z 818.328,A -85,B 0,C 180,E1 11446.01,E2 11446.01} C_VEL
LIN {X 0,Y 217.416,Z 823.253,A -85,B 0,C 180,E1 11440.868,E2 11440.868} C_VEL
LIN {X 0,Y 218,Z 826.132,A -85,B 0,C 180,E1 11436.319,E2 11436.319} C_VEL
LIN {X 0,Y 218.599,Z 827.503,A -85,B 0,C 180,E1 11432.097,E2 11432.097} C_VEL
LIN {X 0,Y 218.662,Z 827.594,A -85,B 0,C 180,E1 11428.69,E2 11428.69} C_VEL
LIN {X 0,Y 218.175,Z 826.603,A -85,B 0,C 180,E1 11424.741,E2 11424.741} C_VEL
LIN {X 0,Y 217.525,Z 824.016,A -85,B 0,C 180,E1 11420.208,E2 11420.208} C_VEL
LIN {X 0,Y 217.399,Z 819.492,A -85,B 0,C 180,E1 11415.075,E2 11415.075} C_VEL
LIN {X 0,Y 218.362,Z 813.188,A -85,B 0,C 180,E1 11409.915,E2 11409.915} C_VEL
LIN {X 0,Y 220.725,Z 804.999,A -85,B 0,C 180,E1 11404.799,E2 11404.799} C_VEL
LIN {X 0,Y 224.747,Z 794.465,A -85,B 0,C 180,E1 11399.662,E2 11399.662} C_VEL
LIN {X 0,Y 230.05,Z 782.292,A -85,B 0,C 180,E1 11394.992,E2 11394.992} C_VEL
LIN {X 0,Y 236.245,Z 768.859,A -85,B 0,C 180,E1 11390.906,E2 11390.906} C_VEL
LIN {X 0,Y 243.147,Z 753.856,A -85,B 0,C 180,E1 11387.274,E2 11387.274} C_VEL
LIN {X 0,Y 250.279,Z 737.764,A -85,B 0,C 180,E1 11384.186,E2 11384.186} C_VEL
LIN {X 0,Y 257.346,Z 720.677,A -85,B 0,C 180,E1 11381.592,E2 11381.592} C_VEL
LIN {X 0,Y 263.764,Z 703.556,A -85,B 0,C 180,E1 11379.538,E2 11379.538} C_VEL
LIN {X 0,Y 269.728,Z 685.704,A -85,B 0,C 180,E1 11377.857,E2 11377.857} C_VEL
LIN {X 0,Y 275.313,Z 666.188,A -85,B 0,C 180,E1 11376.447,E2 11376.447} C_VEL
LIN {X 0,Y 280.038,Z 645.527,A -85,B 0,C 180,E1 11375.34,E2 11375.34} C_VEL
LIN {X 0,Y 283.464,Z 624.268,A -85,B 0,C 180,E1 11374.508,E2 11374.508} C_VEL
LIN {X 0,Y 285.834,Z 598.19,A -85,B 0,C 180,E1 11373.805,E2 11373.805} C_VEL
LIN {X 0,Y 296.611,Z 450.834,A -85,B 0,C 180,E1 11370.346,E2 11370.346} C_VEL
LIN {X 0,Y 289.027,Z 435.767,A -85,B 0,C 180,E1 11367.282,E2 11367.282} C_VEL
LIN {X 0,Y 282.139,Z 423.569,A -85,B 0,C 180,E1 11364.161,E2 11364.161} C_VEL
LIN {X 0,Y 276.319,Z 414.042,A -85,B 0,C 180,E1 11361.158,E2 11361.158} C_VEL
LIN {X 0,Y 270.063,Z 404.188,A -85,B 0,C 180,E1 11357.339,E2 11357.339} C_VEL
LIN {X 0,Y 265.445,Z 397.664,A -85,B 0,C 180,E1 11353.949,E2 11353.949} C_VEL
LIN {X 0,Y 262.933,Z 394.104,A -85,B 0,C 180,E1 11351.738,E2 11351.738} C_VEL
LIN {X 0,Y 259.698,Z 389.302,A -85,B 0,C 180,E1 11348.189,E2 11348.189} C_VEL
LIN {X 0,Y 256.345,Z 384.467,A -85,B 0,C 180,E1 11342.459,E2 11342.459} C_VEL
LIN {X 0,Y 255.184,Z 383.158,A -85,B 0,C 180,E1 11336.18,E2 11336.18} C_VEL
LIN {X 0,Y 256.707,Z 384.087,A -85,B 0,C 180,E1 11330.132,E2 11330.132} C_VEL
LIN {X 0,Y 257.898,Z 385.192,A -85,B 0,C 180,E1 11327.915,E2 11327.915} C_VEL
LIN {X 0,Y 262.35,Z 390.573,A -85,B 0,C 180,E1 11322.362,E2 11322.362} C_VEL
LIN {X 0,Y 266.721,Z 396.22,A -85,B 0,C 180,E1 11318.561,E2 11318.561} C_VEL
LIN {X 0,Y 270.799,Z 401.697,A -85,B 0,C 180,E1 11315.689,E2 11315.689} C_VEL
LIN {X 0,Y 274.657,Z 407.011,A -85,B 0,C 180,E1 11313.341,E2 11313.341} C_VEL
LIN {X 0,Y 279.64,Z 414.192,A -85,B 0,C 180,E1 11310.669,E2 11310.669} C_VEL
LIN {X 0,Y 286.222,Z 424.561,A -85,B 0,C 180,E1 11307.573,E2 11307.573} C_VEL
LIN {X 0,Y 293.136,Z 436.486,A -85,B 0,C 180,E1 11304.709,E2 11304.709} C_VEL
LIN {X 0,Y 296.121,Z 442.35,A -85,B 0,C 180,E1 11303.551,E2 11303.551} C_VEL
LIN {X 0,Y 287.45,Z 575.037,A -85,B 0,C 180,E1 11300.618,E2 11300.618} C_VEL
LIN {X 0,Y 285.615,Z 594.636,A -85,B 0,C 180,E1 11299.909,E2 11299.909} C_VEL
LIN {X 0,Y 282.763,Z 613.24,A -85,B 0,C 180,E1 11298.941,E2 11298.941} C_VEL
LIN {X 0,Y 278.956,Z 631.262,A -85,B 0,C 180,E1 11297.684,E2 11297.684} C_VEL
LIN {X 0,Y 274.431,Z 648.157,A -85,B 0,C 180,E1 11296.168,E2 11296.168} C_VEL
LIN {X 0,Y 269.082,Z 664.6,A -85,B 0,C 180,E1 11294.311,E2 11294.311} C_VEL
LIN {X 0,Y 262.908,Z 680.715,A -85,B 0,C 180,E1 11292.015,E2 11292.015} C_VEL
LIN {X 0,Y 256.578,Z 695.169,A -85,B 0,C 180,E1 11289.433,E2 11289.433} C_VEL
LIN {X 0,Y 249.799,Z 708.983,A -85,B 0,C 180,E1 11286.326,E2 11286.326} C_VEL
LIN {X 0,Y 243.239,Z 721.158,A -85,B 0,C 180,E1 11282.86,E2 11282.86} C_VEL
LIN {X 0,Y 237.107,Z 731.773,A -85,B 0,C 180,E1 11279.008,E2 11279.008} C_VEL
LIN {X 0,Y 231.628,Z 740.837,A -85,B 0,C 180,E1 11274.753,E2 11274.753} C_VEL
LIN {X 0,Y 226.97,Z 748.334,A -85,B 0,C 180,E1 11270.096,E2 11270.096} C_VEL
LIN {X 0,Y 223.517,Z 753.966,A -85,B 0,C 180,E1 11265.303,E2 11265.303} C_VEL
LIN {X 0,Y 221.088,Z 758.053,A -85,B 0,C 180,E1 11260.158,E2 11260.158} C_VEL
LIN {X 0,Y 219.761,Z 760.419,A -85,B 0,C 180,E1 11254.959,E2 11254.959} C_VEL
LIN {X 0,Y 219.383,Z 761.161,A -85,B 0,C 180,E1 11249.739,E2 11249.739} C_VEL
LIN {X 0,Y 219.84,Z 760.314,A -85,B 0,C 180,E1 11244.52,E2 11244.52} C_VEL
LIN {X 0,Y 221.255,Z 757.829,A -85,B 0,C 180,E1 11239.323,E2 11239.323} C_VEL
LIN {X 0,Y 223.781,Z 753.598,A -85,B 0,C 180,E1 11234.184,E2 11234.184} C_VEL
LIN {X 0,Y 227.562,Z 747.464,A -85,B 0,C 180,E1 11229.152,E2 11229.152} C_VEL
LIN {X 0,Y 232.39,Z 739.694,A -85,B 0,C 180,E1 11224.517,E2 11224.517} C_VEL
LIN {X 0,Y 237.688,Z 730.931,A -85,B 0,C 180,E1 11220.518,E2 11220.518} C_VEL
LIN {X 0,Y 243.916,Z 720.117,A -85,B 0,C 180,E1 11216.683,E2 11216.683} C_VEL
LIN {X 0,Y 250.552,Z 707.71,A -85,B 0,C 180,E1 11213.232,E2 11213.232} C_VEL
LIN {X 0,Y 257.163,Z 694.13,A -85,B 0,C 180,E1 11210.241,E2 11210.241} C_VEL
LIN {X 0,Y 263.541,Z 679.487,A -85,B 0,C 180,E1 11207.67,E2 11207.67} C_VEL
LIN {X 0,Y 269.486,Z 663.857,A -85,B 0,C 180,E1 11205.475,E2 11205.475} C_VEL
LIN {X 0,Y 275.126,Z 646.327,A -85,B 0,C 180,E1 11203.531,E2 11203.531} C_VEL
LIN {X 0,Y 279.779,Z 628.546,A -85,B 0,C 180,E1 11201.985,E2 11201.985} C_VEL
LIN {X 0,Y 283.603,Z 609.532,A -85,B 0,C 180,E1 11200.724,E2 11200.724} C_VEL
LIN {X 0,Y 286.324,Z 590.113,A -85,B 0,C 180,E1 11199.782,E2 11199.782} C_VEL
LIN {X 0,Y 287.927,Z 569.881,A -85,B 0,C 180,E1 11199.124,E2 11199.124} C_VEL
LIN {X 0,Y 296.194,Z 442.051,A -85,B 0,C 180,E1 11196.301,E2 11196.301} C_VEL
LIN {X 0,Y 289.578,Z 430.115,A -85,B 0,C 180,E1 11193.685,E2 11193.685} C_VEL
LIN {X 0,Y 282.871,Z 419.072,A -85,B 0,C 180,E1 11190.715,E2 11190.715} C_VEL
LIN {X 0,Y 276.297,Z 409.138,A -85,B 0,C 180,E1 11187.361,E2 11187.361} C_VEL
LIN {X 0,Y 272.076,Z 403.378,A -85,B 0,C 180,E1 11184.884,E2 11184.884} C_VEL
LIN {X 0,Y 269.172,Z 399.4,A -85,B 0,C 180,E1 11182.957,E2 11182.957} C_VEL
LIN {X 0,Y 265.748,Z 394.853,A -85,B 0,C 180,E1 11180.367,E2 11180.367} C_VEL
LIN {X 0,Y 261.743,Z 389.755,A -85,B 0,C 180,E1 11176.649,E2 11176.649} C_VEL
LIN {X 0,Y 261.183,Z 389.307,A -85,B 0,C 180,E1 11176.067,E2 11176.067} C_VEL
LIN {X 0,Y 259.511,Z 388.941,A -85,B 0,C 180,E1 11174.267,E2 11174.267} C_VEL
LIN {X 0,Y 255.675,Z 391.866,A -85,B 0,C 180,E1 11168.992,E2 11168.992} C_VEL
LIN {X 0,Y 255.366,Z 391.84,A -85,B 0,C 180,E1 11168.238,E2 11168.238} C_VEL
LIN {X 0,Y 254.495,Z 391.444,A -85,B 0,C 180,E1 11162.477,E2 11162.477} C_VEL
LIN {X 0,Y 255.648,Z 392.802,A -85,B 0,C 180,E1 11157.423,E2 11157.423} C_VEL
LIN {X 0,Y 259,Z 397.844,A -85,B 0,C 180,E1 11151.677,E2 11151.677} C_VEL
LIN {X 0,Y 262.804,Z 403.617,A -85,B 0,C 180,E1 11147.587,E2 11147.587} C_VEL
LIN {X 0,Y 265.841,Z 408.235,A -85,B 0,C 180,E1 11145.015,E2 11145.015} C_VEL
LIN {X 0,Y 269.328,Z 413.494,A -85,B 0,C 180,E1 11142.5,E2 11142.5} C_VEL
LIN {X 0,Y 274.561,Z 421.92,A -85,B 0,C 180,E1 11139.259,E2 11139.259} C_VEL
LIN {X 0,Y 280.356,Z 431.69,A -85,B 0,C 180,E1 11136.179,E2 11136.179} C_VEL
LIN {X 0,Y 286.717,Z 443.639,A -85,B 0,C 180,E1 11133.182,E2 11133.182} C_VEL
LIN {X 0,Y 292.164,Z 454.872,A -85,B 0,C 180,E1 11130.862,E2 11130.862} C_VEL
LIN {X 0,Y 279.571,Z 617.839,A -85,B 0,C 180,E1 11127.02,E2 11127.02} C_VEL
LIN {X 0,Y 276.387,Z 639.389,A -85,B 0,C 180,E1 11126.249,E2 11126.249} C_VEL
LIN {X 0,Y 271.967,Z 659.718,A -85,B 0,C 180,E1 11125.25,E2 11125.25} C_VEL
LIN {X 0,Y 266.475,Z 679.3,A -85,B 0,C 180,E1 11123.956,E2 11123.956} C_VEL
LIN {X 0,Y 260.254,Z 697.966,A -85,B 0,C 180,E1 11122.316,E2 11122.316} C_VEL
LIN {X 0,Y 253.455,Z 715.829,A -85,B 0,C 180,E1 11120.285,E2 11120.285} C_VEL
LIN {X 0,Y 246.249,Z 732.855,A -85,B 0,C 180,E1 11117.816,E2 11117.816} C_VEL
LIN {X 0,Y 238.937,Z 748.793,A -85,B 0,C 180,E1 11114.894,E2 11114.894} C_VEL
LIN {X 0,Y 232.005,Z 763.19,A -85,B 0,C 180,E1 11111.58,E2 11111.58} C_VEL
LIN {X 0,Y 225.452,Z 776.562,A -85,B 0,C 180,E1 11107.734,E2 11107.734} C_VEL
LIN {X 0,Y 219.696,Z 788.576,A -85,B 0,C 180,E1 11103.413,E2 11103.413} C_VEL
LIN {X 0,Y 215.016,Z 799.192,A -85,B 0,C 180,E1 11098.617,E2 11098.617} C_VEL
LIN {X 0,Y 211.658,Z 808.331,A -85,B 0,C 180,E1 11093.378,E2 11093.378} C_VEL
LIN {X 0,Y 209.773,Z 815.863,A -85,B 0,C 180,E1 11087.76,E2 11087.76} C_VEL
LIN {X 0,Y 209.373,Z 821.127,A -85,B 0,C 180,E1 11082.409,E2 11082.409} C_VEL
LIN {X 0,Y 209.898,Z 824.487,A -85,B 0,C 180,E1 11077.389,E2 11077.389} C_VEL
LIN {X 0,Y 210.577,Z 826.182,A -85,B 0,C 180,E1 11072.994,E2 11072.994} C_VEL
LIN {X 0,Y 210.778,Z 826.448,A -85,B 0,C 180,E1 11069.185,E2 11069.185} C_VEL
LIN {X 0,Y 210.346,Z 825.659,A -85,B 0,C 180,E1 11065.365,E2 11065.365} C_VEL
LIN {X 0,Y 209.626,Z 823.367,A -85,B 0,C 180,E1 11060.667,E2 11060.667} C_VEL
LIN {X 0,Y 209.41,Z 819.115,A -85,B 0,C 180,E1 11055.342,E2 11055.342} C_VEL
LIN {X 0,Y 210.328,Z 813.021,A -85,B 0,C 180,E1 11049.985,E2 11049.985} C_VEL
LIN {X 0,Y 212.703,Z 805.097,A -85,B 0,C 180,E1 11044.675,E2 11044.675} C_VEL
LIN {X 0,Y 216.415,Z 795.766,A -85,B 0,C 180,E1 11039.763,E2 11039.763} C_VEL
LIN {X 0,Y 221.57,Z 784.454,A -85,B 0,C 180,E1 11035.034,E2 11035.034} C_VEL
LIN {X 0,Y 227.784,Z 771.682,A -85,B 0,C 180,E1 11030.797,E2 11030.797} C_VEL
LIN {X 0,Y 234.715,Z 757.432,A -85,B 0,C 180,E1 11027.034,E2 11027.034} C_VEL
LIN {X 0,Y 241.925,Z 742.23,A -85,B 0,C 180,E1 11023.848,E2 11023.848} C_VEL
LIN {X 0,Y 249.028,Z 726.281,A -85,B 0,C 180,E1 11021.182,E2 11021.182} C_VEL
LIN {X 0,Y 256.166,Z 708.698,A -85,B 0,C 180,E1 11018.862,E2 11018.862} C_VEL
LIN {X 0,Y 262.822,Z 690.255,A -85,B 0,C 180,E1 11016.976,E2 11016.976} C_VEL
LIN {X 0,Y 268.896,Z 670.685,A -85,B 0,C 180,E1 11015.455,E2 11015.455} C_VEL
LIN {X 0,Y 274.036,Z 650.32,A -85,B 0,C 180,E1 11014.276,E2 11014.276} C_VEL
LIN {X 0,Y 277.885,Z 629.512,A -85,B 0,C 180,E1 11013.388,E2 11013.388} C_VEL
LIN {X 0,Y 280.301,Z 608.505,A -85,B 0,C 180,E1 11012.751,E2 11012.751} C_VEL
LIN {X 0,Y 291.986,Z 454.521,A -85,B 0,C 180,E1 11009.131,E2 11009.131} C_VEL
LIN {X 0,Y 285.192,Z 440.776,A -85,B 0,C 180,E1 11006.215,E2 11006.215} C_VEL
LIN {X 0,Y 278.763,Z 429.163,A -85,B 0,C 180,E1 11003.125,E2 11003.125} C_VEL
LIN {X 0,Y 272.711,Z 418.917,A -85,B 0,C 180,E1 10999.768,E2 10999.768} C_VEL
LIN {X 0,Y 267.395,Z 410.591,A -85,B 0,C 180,E1 10996.286,E2 10996.286} C_VEL
LIN {X 0,Y 263.81,Z 405.188,A -85,B 0,C 180,E1 10993.479,E2 10993.479} C_VEL
LIN {X 0,Y 261.382,Z 401.648,A -85,B 0,C 180,E1 10991.249,E2 10991.249} C_VEL
LIN {X 0,Y 258.367,Z 397.007,A -85,B 0,C 180,E1 10987.784,E2 10987.784} C_VEL
LIN {X 0,Y 255.278,Z 392.346,A -85,B 0,C 180,E1 10982.244,E2 10982.244} C_VEL
LIN {X 0,Y 254.211,Z 391.099,A -85,B 0,C 180,E1 10976.166,E2 10976.166} C_VEL
LIN {X 0,Y 255.704,Z 392.024,A -85,B 0,C 180,E1 10970.18,E2 10970.18} C_VEL
LIN {X 0,Y 256.735,Z 393.017,A -85,B 0,C 180,E1 10968.201,E2 10968.201} C_VEL
LIN {X 0,Y 260.957,Z 398.313,A -85,B 0,C 180,E1 10962.725,E2 10962.725} C_VEL
LIN {X 0,Y 265.1,Z 403.811,A -85,B 0,C 180,E1 10959.003,E2 10959.003} C_VEL
LIN {X 0,Y 268.996,Z 409.205,A -85,B 0,C 180,E1 10956.157,E2 10956.157} C_VEL
LIN {X 0,Y 272.766,Z 414.545,A -85,B 0,C 180,E1 10953.787,E2 10953.787} C_VEL
LIN {X 0,Y 278.112,Z 422.513,A -85,B 0,C 180,E1 10950.846,E2 10950.846} C_VEL
LIN {X 0,Y 284.616,Z 433.283,A -85,B 0,C 180,E1 10947.725,E2 10947.725} C_VEL
LIN {X 0,Y 290.508,Z 443.893,A -85,B 0,C 180,E1 10945.216,E2 10945.216} C_VEL
LIN {X 0,Y 291.54,Z 446.205,A -85,B 0,C 180,E1 10944.786,E2 10944.786} C_VEL
LIN {X 0,Y 282.742,Z 575.597,A -85,B 0,C 180,E1 10941.913,E2 10941.913} C_VEL
LIN {X 0,Y 280.872,Z 595,A -85,B 0,C 180,E1 10941.213,E2 10941.213} C_VEL
LIN {X 0,Y 277.943,Z 613.625,A -85,B 0,C 180,E1 10940.249,E2 10940.249} C_VEL
LIN {X 0,Y 274.124,Z 631.298,A -85,B 0,C 180,E1 10939.026,E2 10939.026} C_VEL
LIN {X 0,Y 269.323,Z 648.727,A -85,B 0,C 180,E1 10937.469,E2 10937.469} C_VEL
LIN {X 0,Y 263.643,Z 665.595,A -85,B 0,C 180,E1 10935.557,E2 10935.557} C_VEL
LIN {X 0,Y 257.362,Z 681.441,A -85,B 0,C 180,E1 10933.29,E2 10933.29} C_VEL
LIN {X 0,Y 250.524,Z 696.445,A -85,B 0,C 180,E1 10930.581,E2 10930.581} C_VEL
LIN {X 0,Y 243.924,Z 709.41,A -85,B 0,C 180,E1 10927.643,E2 10927.643} C_VEL
LIN {X 0,Y 237.034,Z 721.716,A -85,B 0,C 180,E1 10924.125,E2 10924.125} C_VEL
LIN {X 0,Y 230.56,Z 732.446,A -85,B 0,C 180,E1 10920.201,E2 10920.201} C_VEL
LIN {X 0,Y 224.744,Z 741.619,A -85,B 0,C 180,E1 10915.848,E2 10915.848} C_VEL
LIN {X 0,Y 219.767,Z 749.217,A -85,B 0,C 180,E1 10911.064,E2 10911.064} C_VEL
LIN {X 0,Y 215.877,Z 755.172,A -85,B 0,C 180,E1 10905.858,E2 10905.858} C_VEL
LIN {X 0,Y 213.295,Z 759.256,A -85,B 0,C 180,E1 10900.534,E2 10900.534} C_VEL
LIN {X 0,Y 211.878,Z 761.621,A -85,B 0,C 180,E1 10895.144,E2 10895.144} C_VEL
LIN {X 0,Y 211.474,Z 762.363,A -85,B 0,C 180,E1 10889.729,E2 10889.729} C_VEL
LIN {X 0,Y 211.963,Z 761.516,A -85,B 0,C 180,E1 10884.315,E2 10884.315} C_VEL
LIN {X 0,Y 213.473,Z 759.033,A -85,B 0,C 180,E1 10878.929,E2 10878.929} C_VEL
LIN {X 0,Y 216.16,Z 754.805,A -85,B 0,C 180,E1 10873.611,E2 10873.611} C_VEL
LIN {X 0,Y 220.164,Z 748.675,A -85,B 0,C 180,E1 10868.417,E2 10868.417} C_VEL
LIN {X 0,Y 225.254,Z 740.91,A -85,B 0,C 180,E1 10863.649,E2 10863.649} C_VEL
LIN {X 0,Y 230.836,Z 732.13,A -85,B 0,C 180,E1 10859.539,E2 10859.539} C_VEL
LIN {X 0,Y 237.338,Z 721.355,A -85,B 0,C 180,E1 10855.633,E2 10855.633} C_VEL
LIN {X 0,Y 244.262,Z 708.968,A -85,B 0,C 180,E1 10852.121,E2 10852.121} C_VEL
LIN {X 0,Y 251.141,Z 695.418,A -85,B 0,C 180,E1 10849.088,E2 10849.088} C_VEL
LIN {X 0,Y 257.684,Z 681.008,A -85,B 0,C 180,E1 10846.519,E2 10846.519} C_VEL
LIN {X 0,Y 263.925,Z 665.23,A -85,B 0,C 180,E1 10844.276,E2 10844.276} C_VEL
LIN {X 0,Y 269.696,Z 648.035,A -85,B 0,C 180,E1 10842.342,E2 10842.342} C_VEL
LIN {X 0,Y 274.583,Z 630.145,A -85,B 0,C 180,E1 10840.766,E2 10840.766} C_VEL
LIN {X 0,Y 278.565,Z 611.282,A -85,B 0,C 180,E1 10839.495,E2 10839.495} C_VEL
LIN {X 0,Y 281.476,Z 591.614,A -85,B 0,C 180,E1 10838.524,E2 10838.524} C_VEL
LIN {X 0,Y 283.188,Z 571.365,A -85,B 0,C 180,E1 10837.853,E2 10837.853} C_VEL
LIN {X 0,Y 291.6,Z 445.773,A -85,B 0,C 180,E1 10835.054,E2 10835.054} C_VEL
LIN {X 0,Y 285.244,Z 434.181,A -85,B 0,C 180,E1 10832.369,E2 10832.369} C_VEL
LIN {X 0,Y 278.341,Z 422.75,A -85,B 0,C 180,E1 10829.068,E2 10829.068} C_VEL
LIN {X 0,Y 272.996,Z 414.791,A -85,B 0,C 180,E1 10826.131,E2 10826.131} C_VEL
LIN {X 0,Y 269.694,Z 410.128,A -85,B 0,C 180,E1 10824.068,E2 10824.068} C_VEL
LIN {X 0,Y 267.051,Z 406.445,A -85,B 0,C 180,E1 10822.22,E2 10822.22} C_VEL
LIN {X 0,Y 264.021,Z 402.301,A -85,B 0,C 180,E1 10819.813,E2 10819.813} C_VEL
LIN {X 0,Y 260.323,Z 397.438,A -85,B 0,C 180,E1 10816.223,E2 10816.223} C_VEL
LIN {X 0,Y 256.394,Z 392.491,A -85,B 0,C 180,E1 10810.562,E2 10810.562} C_VEL
LIN {X 0,Y 255.366,Z 391.84,A -85,B 0,C 180,E1 10808.238,E2 10808.238} C_VEL
LIN {X 0,Y 254.732,Z 392.537,A -85,B 0,C 180,E1 10806.507,E2 10806.507} C_VEL
LIN {X 0,Y 253.646,Z 399.134,A -85,B 0,C 180,E1 10801.539,E2 10801.539} C_VEL
LIN {X 0,Y 253.773,Z 399.758,A -85,B 0,C 180,E1 10800.41,E2 10800.41} C_VEL
LIN {X 0,Y 254.615,Z 400.805,A -85,B 0,C 180,E1 10797.525,E2 10797.525} C_VEL
LIN {X 0,Y 257.746,Z 405.701,A -85,B 0,C 180,E1 10791.973,E2 10791.973} C_VEL
LIN {X 0,Y 261.341,Z 411.329,A -85,B 0,C 180,E1 10787.965,E2 10787.965} C_VEL
LIN {X 0,Y 264.167,Z 415.792,A -85,B 0,C 180,E1 10785.478,E2 10785.478} C_VEL
LIN {X 0,Y 267.41,Z 420.849,A -85,B 0,C 180,E1 10783.044,E2 10783.044} C_VEL
LIN {X 0,Y 272.569,Z 429.455,A -85,B 0,C 180,E1 10779.718,E2 10779.718} C_VEL
LIN {X 0,Y 278.205,Z 439.428,A -85,B 0,C 180,E1 10776.601,E2 10776.601} C_VEL
LIN {X 0,Y 284.489,Z 451.717,A -85,B 0,C 180,E1 10773.547,E2 10773.547} C_VEL
LIN {X 0,Y 287.648,Z 458.573,A -85,B 0,C 180,E1 10772.124,E2 10772.124} C_VEL
LIN {X 0,Y 275.001,Z 617.004,A -85,B 0,C 180,E1 10768.391,E2 10768.391} C_VEL
LIN {X 0,Y 271.733,Z 638.516,A -85,B 0,C 180,E1 10767.623,E2 10767.623} C_VEL
LIN {X 0,Y 267.063,Z 659.339,A -85,B 0,C 180,E1 10766.602,E2 10766.602} C_VEL
LIN {X 0,Y 261.417,Z 678.827,A -85,B 0,C 180,E1 10765.316,E2 10765.316} C_VEL
LIN {X 0,Y 254.677,Z 698.31,A -85,B 0,C 180,E1 10763.591,E2 10763.591} C_VEL
LIN {X 0,Y 247.356,Z 716.687,A -85,B 0,C 180,E1 10761.457,E2 10761.457} C_VEL
LIN {X 0,Y 239.635,Z 734.022,A -85,B 0,C 180,E1 10758.86,E2 10758.86} C_VEL
LIN {X 0,Y 231.751,Z 750.309,A -85,B 0,C 180,E1 10755.739,E2 10755.739} C_VEL
LIN {X 0,Y 224.017,Z 765.478,A -85,B 0,C 180,E1 10752.027,E2 10752.027} C_VEL
LIN {X 0,Y 216.978,Z 779.045,A -85,B 0,C 180,E1 10747.797,E2 10747.797} C_VEL
LIN {X 0,Y 211.224,Z 790.432,A -85,B 0,C 180,E1 10743.304,E2 10743.304} C_VEL
LIN {X 0,Y 206.527,Z 800.636,A -85,B 0,C 180,E1 10738.224,E2 10738.224} C_VEL
LIN {X 0,Y 203.355,Z 809.086,A -85,B 0,C 180,E1 10732.856,E2 10732.856} C_VEL
LIN {X 0,Y 201.67,Z 816.12,A -85,B 0,C 180,E1 10727.008,E2 10727.008} C_VEL
LIN {X 0,Y 201.462,Z 820.977,A -85,B 0,C 180,E1 10721.45,E2 10721.45} C_VEL
LIN {X 0,Y 202.086,Z 823.833,A -85,B 0,C 180,E1 10716.534,E2 10716.534} C_VEL
LIN {X 0,Y 202.75,Z 825.094,A -85,B 0,C 180,E1 10712.261,E2 10712.261} C_VEL
LIN {X 0,Y 202.849,Z 825.217,A -85,B 0,C 180,E1 10708.87,E2 10708.87} C_VEL
LIN {X 0,Y 202.339,Z 824.355,A -85,B 0,C 180,E1 10704.897,E2 10704.897} C_VEL
LIN {X 0,Y 201.598,Z 821.938,A -85,B 0,C 180,E1 10700.004,E2 10700.004} C_VEL
LIN {X 0,Y 201.499,Z 817.583,A -85,B 0,C 180,E1 10694.458,E2 10694.458} C_VEL
LIN {X 0,Y 202.768,Z 811.047,A -85,B 0,C 180,E1 10688.599,E2 10688.599} C_VEL
LIN {X 0,Y 205.767,Z 802.444,A -85,B 0,C 180,E1 10682.822,E2 10682.822} C_VEL
LIN {X 0,Y 210.348,Z 792.203,A -85,B 0,C 180,E1 10677.513,E2 10677.513} C_VEL
LIN {X 0,Y 216.315,Z 780.23,A -85,B 0,C 180,E1 10672.657,E2 10672.657} C_VEL
LIN {X 0,Y 223.133,Z 767.029,A -85,B 0,C 180,E1 10668.445,E2 10668.445} C_VEL
LIN {X 0,Y 230.465,Z 752.665,A -85,B 0,C 180,E1 10664.821,E2 10664.821} C_VEL
LIN {X 0,Y 237.92,Z 737.371,A -85,B 0,C 180,E1 10661.762,E2 10661.762} C_VEL
LIN {X 0,Y 245.336,Z 721.033,A -85,B 0,C 180,E1 10659.175,E2 10659.175} C_VEL
LIN {X 0,Y 252.706,Z 703.05,A -85,B 0,C 180,E1 10656.945,E2 10656.945} C_VEL
LIN {X 0,Y 259.56,Z 683.999,A -85,B 0,C 180,E1 10655.133,E2 10655.133} C_VEL
LIN {X 0,Y 265.618,Z 664.057,A -85,B 0,C 180,E1 10653.708,E2 10653.708} C_VEL
LIN {X 0,Y 270.646,Z 643.104,A -85,B 0,C 180,E1 10652.605,E2 10652.605} C_VEL
LIN {X 0,Y 274.215,Z 621.815,A -85,B 0,C 180,E1 10651.787,E2 10651.787} C_VEL
LIN {X 0,Y 276.809,Z 594.278,A -85,B 0,C 180,E1 10651.056,E2 10651.056} C_VEL
LIN {X 0,Y 287.438,Z 458.04,A -85,B 0,C 180,E1 10647.85,E2 10647.85} C_VEL
LIN {X 0,Y 280.492,Z 443.907,A -85,B 0,C 180,E1 10644.649,E2 10644.649} C_VEL
LIN {X 0,Y 274.522,Z 432.916,A -85,B 0,C 180,E1 10641.527,E2 10641.527} C_VEL
LIN {X 0,Y 269.085,Z 423.759,A -85,B 0,C 180,E1 10638.243,E2 10638.243} C_VEL
LIN {X 0,Y 265.374,Z 417.733,A -85,B 0,C 180,E1 10635.628,E2 10635.628} C_VEL
LIN {X 0,Y 261.94,Z 412.365,A -85,B 0,C 180,E1 10632.79,E2 10632.79} C_VEL
LIN {X 0,Y 259.84,Z 409.19,A -85,B 0,C 180,E1 10630.756,E2 10630.756} C_VEL
LIN {X 0,Y 257.045,Z 404.709,A -85,B 0,C 180,E1 10627.375,E2 10627.375} C_VEL
LIN {X 0,Y 254.133,Z 400.146,A -85,B 0,C 180,E1 10621.803,E2 10621.803} C_VEL
LIN {X 0,Y 253.248,Z 399.042,A -85,B 0,C 180,E1 10615.924,E2 10615.924} C_VEL
LIN {X 0,Y 254.781,Z 400.014,A -85,B 0,C 180,E1 10610.056,E2 10610.056} C_VEL
LIN {X 0,Y 255.635,Z 400.962,A -85,B 0,C 180,E1 10608.379,E2 10608.379} C_VEL
LIN {X 0,Y 259.582,Z 406.049,A -85,B 0,C 180,E1 10603.093,E2 10603.093} C_VEL
LIN {X 0,Y 263.494,Z 411.398,A -85,B 0,C 180,E1 10599.451,E2 10599.451} C_VEL
LIN {X 0,Y 267.138,Z 416.597,A -85,B 0,C 180,E1 10596.683,E2 10596.683} C_VEL
LIN {X 0,Y 270.805,Z 421.953,A -85,B 0,C 180,E1 10594.289,E2 10594.289} C_VEL
LIN {X 0,Y 276.412,Z 430.661,A -85,B 0,C 180,E1 10591.112,E2 10591.112} C_VEL
LIN {X 0,Y 282.804,Z 441.7,A -85,B 0,C 180,E1 10587.972,E2 10587.972} C_VEL
LIN {X 0,Y 287.099,Z 449.953,A -85,B 0,C 180,E1 10586.061,E2 10586.061} C_VEL
LIN {X 0,Y 278.175,Z 576.264,A -85,B 0,C 180,E1 10583.248,E2 10583.248} C_VEL
LIN {X 0,Y 276.24,Z 595.642,A -85,B 0,C 180,E1 10582.549,E2 10582.549} C_VEL
LIN {X 0,Y 273.3,Z 613.874,A -85,B 0,C 180,E1 10581.61,E2 10581.61} C_VEL
LIN {X 0,Y 269.208,Z 632.219,A -85,B 0,C 180,E1 10580.343,E2 10580.343} C_VEL
LIN {X 0,Y 264.064,Z 650.173,A -85,B 0,C 180,E1 10578.728,E2 10578.728} C_VEL
LIN {X 0,Y 258.321,Z 666.619,A -85,B 0,C 180,E1 10576.852,E2 10576.852} C_VEL
LIN {X 0,Y 251.676,Z 682.752,A -85,B 0,C 180,E1 10574.522,E2 10574.522} C_VEL
LIN {X 0,Y 244.577,Z 697.719,A -85,B 0,C 180,E1 10571.785,E2 10571.785} C_VEL
LIN {X 0,Y 237.236,Z 711.482,A -85,B 0,C 180,E1 10568.59,E2 10568.59} C_VEL
LIN {X 0,Y 230.094,Z 723.622,A -85,B 0,C 180,E1 10565,E2 10565} C_VEL
LIN {X 0,Y 223.373,Z 734.214,A -85,B 0,C 180,E1 10560.981,E2 10560.981} C_VEL
LIN {X 0,Y 217.322,Z 743.265,A -85,B 0,C 180,E1 10556.504,E2 10556.504} C_VEL
LIN {X 0,Y 212.138,Z 750.752,A -85,B 0,C 180,E1 10551.569,E2 10551.569} C_VEL
LIN {X 0,Y 208.258,Z 756.378,A -85,B 0,C 180,E1 10546.455,E2 10546.455} C_VEL
LIN {X 0,Y 205.511,Z 760.46,A -85,B 0,C 180,E1 10540.938,E2 10540.938} C_VEL
LIN {X 0,Y 203.998,Z 762.823,A -85,B 0,C 180,E1 10535.343,E2 10535.343} C_VEL
LIN {X 0,Y 203.564,Z 763.564,A -85,B 0,C 180,E1 10529.719,E2 10529.719} C_VEL
LIN {X 0,Y 204.088,Z 762.719,A -85,B 0,C 180,E1 10524.095,E2 10524.095} C_VEL
LIN {X 0,Y 205.702,Z 760.237,A -85,B 0,C 180,E1 10518.505,E2 10518.505} C_VEL
LIN {X 0,Y 208.562,Z 756.013,A -85,B 0,C 180,E1 10512.997,E2 10512.997} C_VEL
LIN {X 0,Y 212.806,Z 749.886,A -85,B 0,C 180,E1 10507.631,E2 10507.631} C_VEL
LIN {X 0,Y 218.173,Z 742.127,A -85,B 0,C 180,E1 10502.724,E2 10502.724} C_VEL
LIN {X 0,Y 224.187,Z 733.116,A -85,B 0,C 180,E1 10498.414,E2 10498.414} C_VEL
LIN {X 0,Y 230.874,Z 722.544,A -85,B 0,C 180,E1 10494.508,E2 10494.508} C_VEL
LIN {X 0,Y 238.068,Z 710.226,A -85,B 0,C 180,E1 10490.953,E2 10490.953} C_VEL
LIN {X 0,Y 245.027,Z 697.109,A -85,B 0,C 180,E1 10487.96,E2 10487.96} C_VEL
LIN {X 0,Y 251.826,Z 682.732,A -85,B 0,C 180,E1 10485.352,E2 10485.352} C_VEL
LIN {X 0,Y 258.482,Z 666.589,A -85,B 0,C 180,E1 10483.024,E2 10483.024} C_VEL
LIN {X 0,Y 264.53,Z 649.256,A -85,B 0,C 180,E1 10481.059,E2 10481.059} C_VEL
LIN {X 0,Y 269.81,Z 630.562,A -85,B 0,C 180,E1 10479.409,E2 10479.409} C_VEL
LIN {X 0,Y 273.95,Z 611.411,A -85,B 0,C 180,E1 10478.129,E2 10478.129} C_VEL
LIN {X 0,Y 276.91,Z 591.815,A -85,B 0,C 180,E1 10477.172,E2 10477.172} C_VEL
LIN {X 0,Y 278.665,Z 571.553,A -85,B 0,C 180,E1 10476.505,E2 10476.505} C_VEL
LIN {X 0,Y 287.196,Z 449.723,A -85,B 0,C 180,E1 10473.791,E2 10473.791} C_VEL
LIN {X 0,Y 281.605,Z 439.42,A -85,B 0,C 180,E1 10471.284,E2 10471.284} C_VEL
LIN {X 0,Y 275.622,Z 429.222,A -85,B 0,C 180,E1 10468.256,E2 10468.256} C_VEL
LIN {X 0,Y 270.553,Z 421.467,A -85,B 0,C 180,E1 10465.326,E2 10465.326} C_VEL
LIN {X 0,Y 265.812,Z 414.52,A -85,B 0,C 180,E1 10462.096,E2 10462.096} C_VEL
LIN {X 0,Y 262.321,Z 409.742,A -85,B 0,C 180,E1 10459.251,E2 10459.251} C_VEL
LIN {X 0,Y 259.022,Z 405.21,A -85,B 0,C 180,E1 10455.907,E2 10455.907} C_VEL
LIN {X 0,Y 255.316,Z 400.383,A -85,B 0,C 180,E1 10450.379,E2 10450.379} C_VEL
LIN {X 0,Y 253.544,Z 399.292,A -85,B 0,C 180,E1 10444.298,E2 10444.298} C_VEL
LIN {X 0,Y 253.773,Z 399.758,A -85,B 0,C 180,E1 10440.41,E2 10440.41} C_VEL
LIN {X 0,Y 254.033,Z 401.002,A -85,B 0,C 180,E1 10438.942,E2 10438.942} C_VEL
LIN {X 0,Y 254.391,Z 405.124,A -85,B 0,C 180,E1 10436.876,E2 10436.876} C_VEL
LIN {X 0,Y 255.3,Z 411.169,A -85,B 0,C 180,E1 10434.154,E2 10434.154} C_VEL
LIN {X 0,Y 256.033,Z 412.675,A -85,B 0,C 180,E1 10432.953,E2 10432.953} C_VEL
LIN {X 0,Y 259.784,Z 418.856,A -85,B 0,C 180,E1 10428.455,E2 10428.455} C_VEL
LIN {X 0,Y 262.574,Z 423.451,A -85,B 0,C 180,E1 10425.895,E2 10425.895} C_VEL
LIN {X 0,Y 265.576,Z 428.32,A -85,B 0,C 180,E1 10423.543,E2 10423.543} C_VEL
LIN {X 0,Y 270.665,Z 437.112,A -85,B 0,C 180,E1 10420.132,E2 10420.132} C_VEL
LIN {X 0,Y 276.337,Z 447.743,A -85,B 0,C 180,E1 10416.885,E2 10416.885} C_VEL
LIN {X 0,Y 282.122,Z 459.501,A -85,B 0,C 180,E1 10413.987,E2 10413.987} C_VEL
LIN {X 0,Y 283.275,Z 462.416,A -85,B 0,C 180,E1 10413.422,E2 10413.422} C_VEL
LIN {X 0,Y 270.604,Z 616.092,A -85,B 0,C 180,E1 10409.809,E2 10409.809} C_VEL
LIN {X 0,Y 267.256,Z 637.577,A -85,B 0,C 180,E1 10409.048,E2 10409.048} C_VEL
LIN {X 0,Y 262.685,Z 657.614,A -85,B 0,C 180,E1 10408.079,E2 10408.079} C_VEL
LIN {X 0,Y 256.869,Z 677.223,A -85,B 0,C 180,E1 10406.81,E2 10406.81} C_VEL
LIN {X 0,Y 250.242,Z 695.894,A -85,B 0,C 180,E1 10405.192,E2 10405.192} C_VEL
LIN {X 0,Y 242.954,Z 713.742,A -85,B 0,C 180,E1 10403.171,E2 10403.171} C_VEL
LIN {X 0,Y 235.181,Z 730.745,A -85,B 0,C 180,E1 10400.691,E2 10400.691} C_VEL
LIN {X 0,Y 227.13,Z 746.833,A -85,B 0,C 180,E1 10397.692,E2 10397.692} C_VEL
LIN {X 0,Y 219.339,Z 761.458,A -85,B 0,C 180,E1 10394.221,E2 10394.221} C_VEL
LIN {X 0,Y 211.672,Z 775.476,A -85,B 0,C 180,E1 10389.97,E2 10389.97} C_VEL
LIN {X 0,Y 204.949,Z 787.885,A -85,B 0,C 180,E1 10385.145,E2 10385.145} C_VEL
LIN {X 0,Y 199.532,Z 798.686,A -85,B 0,C 180,E1 10379.741,E2 10379.741} C_VEL
LIN {X 0,Y 195.73,Z 807.819,A -85,B 0,C 180,E1 10373.8,E2 10373.8} C_VEL
LIN {X 0,Y 193.793,Z 814.866,A -85,B 0,C 180,E1 10367.722,E2 10367.722} C_VEL
LIN {X 0,Y 193.479,Z 819.739,A -85,B 0,C 180,E1 10361.929,E2 10361.929} C_VEL
LIN {X 0,Y 194.102,Z 822.611,A -85,B 0,C 180,E1 10356.804,E2 10356.804} C_VEL
LIN {X 0,Y 194.822,Z 823.889,A -85,B 0,C 180,E1 10352.353,E2 10352.353} C_VEL
LIN {X 0,Y 194.934,Z 824.015,A -85,B 0,C 180,E1 10348.824,E2 10348.824} C_VEL
LIN {X 0,Y 194.421,Z 823.231,A -85,B 0,C 180,E1 10344.985,E2 10344.985} C_VEL
LIN {X 0,Y 193.632,Z 820.899,A -85,B 0,C 180,E1 10339.889,E2 10339.889} C_VEL
LIN {X 0,Y 193.557,Z 816.614,A -85,B 0,C 180,E1 10334.111,E2 10334.111} C_VEL
LIN {X 0,Y 194.953,Z 810.141,A -85,B 0,C 180,E1 10328.014,E2 10328.014} C_VEL
LIN {X 0,Y 197.969,Z 802.088,A -85,B 0,C 180,E1 10322.313,E2 10322.313} C_VEL
LIN {X 0,Y 202.462,Z 792.615,A -85,B 0,C 180,E1 10317.091,E2 10317.091} C_VEL
LIN {X 0,Y 208.492,Z 781.169,A -85,B 0,C 180,E1 10312.133,E2 10312.133} C_VEL
LIN {X 0,Y 215.572,Z 768.227,A -85,B 0,C 180,E1 10307.739,E2 10307.739} C_VEL
LIN {X 0,Y 223.377,Z 753.787,A -85,B 0,C 180,E1 10303.893,E2 10303.893} C_VEL
LIN {X 0,Y 231.624,Z 737.758,A -85,B 0,C 180,E1 10300.56,E2 10300.56} C_VEL
LIN {X 0,Y 239.679,Z 720.833,A -85,B 0,C 180,E1 10297.823,E2 10297.823} C_VEL
LIN {X 0,Y 247.201,Z 703.258,A -85,B 0,C 180,E1 10295.613,E2 10295.613} C_VEL
LIN {X 0,Y 254.038,Z 685.125,A -85,B 0,C 180,E1 10293.856,E2 10293.856} C_VEL
LIN {X 0,Y 260.107,Z 666.247,A -85,B 0,C 180,E1 10292.463,E2 10292.463} C_VEL
LIN {X 0,Y 265.275,Z 646.29,A -85,B 0,C 180,E1 10291.365,E2 10291.365} C_VEL
LIN {X 0,Y 269.18,Z 625.438,A -85,B 0,C 180,E1 10290.515,E2 10290.515} C_VEL
LIN {X 0,Y 271.636,Z 603.776,A -85,B 0,C 180,E1 10289.889,E2 10289.889} C_VEL
LIN {X 0,Y 283.093,Z 461.902,A -85,B 0,C 180,E1 10286.566,E2 10286.566} C_VEL
LIN {X 0,Y 277.185,Z 449.518,A -85,B 0,C 180,E1 10283.659,E2 10283.659} C_VEL
LIN {X 0,Y 271.628,Z 439.041,A -85,B 0,C 180,E1 10280.581,E2 10280.581} C_VEL
LIN {X 0,Y 266.236,Z 429.526,A -85,B 0,C 180,E1 10277.089,E2 10277.089} C_VEL
LIN {X 0,Y 262.995,Z 424.271,A -85,B 0,C 180,E1 10274.644,E2 10274.644} C_VEL
LIN {X 0,Y 260.223,Z 419.713,A -85,B 0,C 180,E1 10272.2,E2 10272.2} C_VEL
LIN {X 0,Y 258.215,Z 416.595,A -85,B 0,C 180,E1 10270.147,E2 10270.147} C_VEL
LIN {X 0,Y 255.73,Z 412.411,A -85,B 0,C 180,E1 10266.961,E2 10266.961} C_VEL
LIN {X 0,Y 253.076,Z 408.03,A -85,B 0,C 180,E1 10261.584,E2 10261.584} C_VEL
LIN {X 0,Y 252.289,Z 406.989,A -85,B 0,C 180,E1 10255.681,E2 10255.681} C_VEL
LIN {X 0,Y 253.926,Z 408.051,A -85,B 0,C 180,E1 10249.793,E2 10249.793} C_VEL
LIN {X 0,Y 254.652,Z 409.134,A -85,B 0,C 180,E1 10248.333,E2 10248.333} C_VEL
LIN {X 0,Y 258.219,Z 413.781,A -85,B 0,C 180,E1 10243.464,E2 10243.464} C_VEL
LIN {X 0,Y 261.959,Z 419.081,A -85,B 0,C 180,E1 10239.85,E2 10239.85} C_VEL
LIN {X 0,Y 265.447,Z 424.21,A -85,B 0,C 180,E1 10237.113,E2 10237.113} C_VEL
LIN {X 0,Y 269.931,Z 430.897,A -85,B 0,C 180,E1 10234.14,E2 10234.14} C_VEL
LIN {X 0,Y 275.966,Z 441,A -85,B 0,C 180,E1 10230.717,E2 10230.717} C_VEL
LIN {X 0,Y 282.464,Z 452.944,A -85,B 0,C 180,E1 10227.539,E2 10227.539} C_VEL
LIN {X 0,Y 282.786,Z 454.005,A -85,B 0,C 180,E1 10227.37,E2 10227.37} C_VEL
LIN {X 0,Y 273.755,Z 577.026,A -85,B 0,C 180,E1 10224.624,E2 10224.624} C_VEL
LIN {X 0,Y 271.752,Z 596.364,A -85,B 0,C 180,E1 10223.925,E2 10223.925} C_VEL
LIN {X 0,Y 268.767,Z 614.358,A -85,B 0,C 180,E1 10223.003,E2 10223.003} C_VEL
LIN {X 0,Y 264.695,Z 632.223,A -85,B 0,C 180,E1 10221.783,E2 10221.783} C_VEL
LIN {X 0,Y 259.577,Z 649.758,A -85,B 0,C 180,E1 10220.23,E2 10220.23} C_VEL
LIN {X 0,Y 253.291,Z 667.268,A -85,B 0,C 180,E1 10218.249,E2 10218.249} C_VEL
LIN {X 0,Y 246.395,Z 683.474,A -85,B 0,C 180,E1 10215.909,E2 10215.909} C_VEL
LIN {X 0,Y 239.01,Z 698.506,A -85,B 0,C 180,E1 10213.154,E2 10213.154} C_VEL
LIN {X 0,Y 231.599,Z 711.922,A -85,B 0,C 180,E1 10210.034,E2 10210.034} C_VEL
LIN {X 0,Y 224.101,Z 724.189,A -85,B 0,C 180,E1 10206.397,E2 10206.397} C_VEL
LIN {X 0,Y 217.005,Z 734.895,A -85,B 0,C 180,E1 10202.307,E2 10202.307} C_VEL
LIN {X 0,Y 210.58,Z 744.05,A -85,B 0,C 180,E1 10197.73,E2 10197.73} C_VEL
LIN {X 0,Y 205.038,Z 751.635,A -85,B 0,C 180,E1 10192.658,E2 10192.658} C_VEL
LIN {X 0,Y 200.85,Z 757.35,A -85,B 0,C 180,E1 10187.378,E2 10187.378} C_VEL
LIN {X 0,Y 197.854,Z 761.519,A -85,B 0,C 180,E1 10181.662,E2 10181.662} C_VEL
LIN {X 0,Y 196.174,Z 763.962,A -85,B 0,C 180,E1 10175.851,E2 10175.851} C_VEL
LIN {X 0,Y 195.656,Z 764.775,A -85,B 0,C 180,E1 10170,E2 10170} C_VEL
LIN {X 0,Y 196.162,Z 763.998,A -85,B 0,C 180,E1 10164.149,E2 10164.149} C_VEL
LIN {X 0,Y 197.823,Z 761.596,A -85,B 0,C 180,E1 10158.336,E2 10158.336} C_VEL
LIN {X 0,Y 200.801,Z 757.468,A -85,B 0,C 180,E1 10152.617,E2 10152.617} C_VEL
LIN {X 0,Y 205.284,Z 751.395,A -85,B 0,C 180,E1 10147.008,E2 10147.008} C_VEL
LIN {X 0,Y 210.828,Z 743.822,A -85,B 0,C 180,E1 10141.998,E2 10141.998} C_VEL
LIN {X 0,Y 217.302,Z 734.606,A -85,B 0,C 180,E1 10137.43,E2 10137.43} C_VEL
LIN {X 0,Y 224.661,Z 723.474,A -85,B 0,C 180,E1 10133.236,E2 10133.236} C_VEL
LIN {X 0,Y 231.984,Z 711.472,A -85,B 0,C 180,E1 10129.719,E2 10129.719} C_VEL
LIN {X 0,Y 239.687,Z 697.456,A -85,B 0,C 180,E1 10126.506,E2 10126.506} C_VEL
LIN {X 0,Y 247.006,Z 682.446,A -85,B 0,C 180,E1 10123.805,E2 10123.805} C_VEL
LIN {X 0,Y 253.758,Z 666.463,A -85,B 0,C 180,E1 10121.529,E2 10121.529} C_VEL
LIN {X 0,Y 259.939,Z 649.121,A -85,B 0,C 180,E1 10119.59,E2 10119.59} C_VEL
LIN {X 0,Y 265.193,Z 630.945,A -85,B 0,C 180,E1 10118.004,E2 10118.004} C_VEL
LIN {X 0,Y 269.4,Z 612.029,A -85,B 0,C 180,E1 10116.746,E2 10116.746} C_VEL
LIN {X 0,Y 272.432,Z 592.635,A -85,B 0,C 180,E1 10115.799,E2 10115.799} C_VEL
LIN {X 0,Y 274.264,Z 572.377,A -85,B 0,C 180,E1 10115.13,E2 10115.13} C_VEL
LIN {X 0,Y 282.882,Z 453.569,A -85,B 0,C 180,E1 10112.467,E2 10112.467} C_VEL
LIN {X 0,Y 276.468,Z 441.753,A -85,B 0,C 180,E1 10109.344,E2 10109.344} C_VEL
LIN {X 0,Y 271.149,Z 432.812,A -85,B 0,C 180,E1 10106.382,E2 10106.382} C_VEL
LIN {X 0,Y 266.347,Z 425.421,A -85,B 0,C 180,E1 10103.273,E2 10103.273} C_VEL
LIN {X 0,Y 263.351,Z 421.042,A -85,B 0,C 180,E1 10101.026,E2 10101.026} C_VEL
LIN {X 0,Y 260.769,Z 417.311,A -85,B 0,C 180,E1 10098.789,E2 10098.789} C_VEL
LIN {X 0,Y 257.678,Z 412.938,A -85,B 0,C 180,E1 10095.53,E2 10095.53} C_VEL
LIN {X 0,Y 254.241,Z 408.276,A -85,B 0,C 180,E1 10090.194,E2 10090.194} C_VEL
LIN {X 0,Y 252.572,Z 407.233,A -85,B 0,C 180,E1 10084.314,E2 10084.314} C_VEL
LIN {X 0,Y 253.333,Z 408.221,A -85,B 0,C 180,E1 10078.417,E2 10078.417} C_VEL
LIN {X 0,Y 256.033,Z 412.675,A -85,B 0,C 180,E1 10072.953,E2 10072.953} C_VEL
LIN {X 0,Y 256.979,Z 414.785,A -85,B 0,C 180,E1 10071.57,E2 10071.57} C_VEL
LIN {X 0,Y 258.033,Z 419.596,A -85,B 0,C 180,E1 10069.915,E2 10069.915} C_VEL
LIN {X 0,Y 259.923,Z 428.541,A -85,B 0,C 180,E1 10067.346,E2 10067.346} C_VEL
LIN {X 0,Y 261.024,Z 431.187,A -85,B 0,C 180,E1 10066.272,E2 10066.272} C_VEL
